(* CODESYS project SmiuUGP_Dubniki.project
   Version: 1.0
   Company: ENTEL

Project tree, tasks and I/O mapping:
  CODESYS_Control_for_Raspberry_Pi : CODESYS Control for Raspberry Pi, 3S - Smart Software Solutions GmbH, version 3.5.8.10
    application Application
      libraries: Util, * (System); AlarmManager, * (Intern); Alarm Manager Interfaces, * (Intern); Standard, * (System); VisuDialogs, * (System)
      task MainTask (cyclic, interval t#50ms, priority 2, watchdog t#1000ms x 1) calls PLC_PRG, GPIO_HANDLER, AlarmChecker
      task VISU_TASK (cyclic, interval 100 ms, priority 30) calls VisuElems.Visu_Prg
      task AlarmManagerTask (cyclic, interval 50 ms, priority 31) calls AlarmManager.Alarm_Prg
      task BusTask (cyclic, interval t#20ms, priority 1, watchdog t#1000ms x 1) calls BusReinit
      program PLC_PRG [ST]
      image pool ImagePool
      program GPIO_HANDLER [ST]
      visualization/
        visualisation monitoring
        ups_s2/
          visualisation ups_s2_state
          visualisation ups_s2_params
        visualisation main
        visualisation info
        visualisation climate
        visualisation alarm
        visualisation schrps
        visualisation shasn
        visualisation logs
        visualisation schrpa
        ups_s1/
          visualisation ups_s1_params
          visualisation ups_s1_state
        ups_a1/
          visualisation ups_a1_params
          visualisation ups_a1_state
        ups_a2/
          visualisation ups_a2_state
          visualisation ups_a2_params
        visualisation climate_log
        visualisation more
      Alarm Configuration
        alarm class Error (priority 10, acknowledge REP)
        alarm class Warning (priority 30, acknowledge REP)
        alarm class Info (priority 100, acknowledge REP)
        AlarmStorage
        text list AlarmGroup
        alarm group AlarmGroup
            93 [Error]: Comparison Equal, ExpressionToCompare TRUE, Expression AlarmChecker.ups_s2_out_v_alarm - "Отсутствует напряжение на выходе ИБП С2"
            94 [Error]: Comparison Equal, ExpressionToCompare TRUE, Expression AlarmChecker.ups_a1_out_v_alarm - "Отсутствует напряжение на выходе ИБП А1"
            49 [Error]: Comparison Equal, ExpressionToCompare TRUE, Expression PLC_PRG.ips_s1_alarm - "Авария ИБП С1"
            103 [Error]: Comparison Equal, ExpressionToCompare FALSE, Expression PLC_PRG.ips_s2_input_present - "ИБП С2 работает от АКБ"
            101 [Error]: Comparison Equal, ExpressionToCompare TRUE, Expression AlarmChecker.shrps_in_2_alarm - "Отсутствует напряжение на резервном вводе ЩРПС"
            97 [Error]: Comparison Equal, ExpressionToCompare TRUE, Expression GPIO_HANDLER.IN_1 - "Нарушение ШОС"
            100 [Error]: Comparison Equal, ExpressionToCompare TRUE, Expression AlarmChecker.shrps_in_1_alarm - "Отсутствует напряжение на основном вводе ЩРПC"
            92 [Error]: Comparison Equal, ExpressionToCompare TRUE, Expression AlarmChecker.ups_s1_out_v_alarm - "Отсутствует напряжение на выходе ИБП С1"
            95 [Error]: Comparison Equal, ExpressionToCompare TRUE, Expression AlarmChecker.ups_a2_out_v_alarm - "Отсутствует напряжение на выходе ИБП А2"
            47 [Error]: Comparison Equal, ExpressionToCompare TRUE, Expression PLC_PRG.ips_a2_alarm - "Авария ИБП А2"
            98 [Error]: Comparison Equal, ExpressionToCompare TRUE, Expression GPIO_HANDLER.IN_3 - "Авария ШОС"
            6 [Error]: Comparison Equal, ExpressionToCompare FALSE, Expression GPIO_HANDLER.IN_6 - "Отсутствует напряжение на шине БП ШАСН"
            90 [Error]: Comparison Equal, ExpressionToCompare TRUE, Expression AlarmChecker.ups_a1_in_v_alarm - "Отсутствует напряжение на входе ИБП А1"
            0 [Error]: Comparison Equal, ExpressionToCompare TRUE, Expression AlarmChecker.shrpa_in_1_alarm - "Отсутствует напряжение на основном вводе ЩРПА"
            1 [Error]: Comparison Equal, ExpressionToCompare TRUE, Expression AlarmChecker.shrpa_in_2_alarm - "Отсутствует напряжение на резервном вводе ЩРПА"
            2 [Error]: Comparison Equal, ExpressionToCompare FALSE, Expression GPIO_HANDLER.IN_4 - "Отсутствует напряжение на основном вводе ШАСН"
            3 [Error]: Comparison Equal, ExpressionToCompare FALSE, Expression GPIO_HANDLER.IN_5 - "Отсутствует напряжение на резервном вводе ШАСН"
            4 [Error]: Comparison Equal, ExpressionToCompare FALSE, Expression PLC_PRG.shrps_ups_bus_1 - "Отсутствует напряжение на ГП 1 ЩРПС"
            5 [Error]: Comparison Equal, ExpressionToCompare FALSE, Expression PLC_PRG.shrps_ups_bus_2 - "Отсутствует напряжение на ГП 2 ЩРПС"
            45 [Error]: Comparison Equal, ExpressionToCompare TRUE, Expression PLC_PRG.ips_a1_alarm - "Авария ИБП А1"
            102 [Error]: Comparison Equal, ExpressionToCompare FALSE, Expression PLC_PRG.ips_s1_input_present - "ИБП С1 работает от АКБ"
            88 [Error]: Comparison Equal, ExpressionToCompare TRUE, Expression AlarmChecker.ups_s1_in_v_alarm - "Отсутствует напряжение на входе ИБП С1"
            89 [Error]: Comparison Equal, ExpressionToCompare TRUE, Expression AlarmChecker.ups_s2_in_v_alarm - "Отсутствует напряжение на входе ИБП С2"
            99 [Error]: Comparison Equal, ExpressionToCompare TRUE, Expression AlarmChecker.shrpa_out_alarm - "Отсутствует напряжение на ШБПА  ЩРПА"
            91 [Error]: Comparison Equal, ExpressionToCompare TRUE, Expression AlarmChecker.ups_a2_in_v_alarm - "Отсутствует напряжение на входе ИБП А2"
            53 [Error]: Comparison Equal, ExpressionToCompare TRUE, Expression PLC_PRG.ips_s2_alarm - "Авария ИБП С2"
            96 [Error]: Comparison Equal, ExpressionToCompare TRUE, Expression GPIO_HANDLER.IN_2 - "Пожар"
            7 [Error]: Comparison Equal, ExpressionToCompare FALSE, Expression GPIO_HANDLER.IN_7 - "Отсутствует напряжение на шине ГП ШАСН"
        text list ClimateGroup
        alarm group ClimateGroup
            8 [Info]: Comparison Equal, ExpressionToCompare TRUE, Expression PLC_PRG.climate_condition_1_state - "Кондиционеры включены"
            11 [Info]: Comparison Equal, ExpressionToCompare FALSE, Expression PLC_PRG.climate_heat_door_state - "Обогрев дверей выключен"
            9 [Info]: Comparison Equal, ExpressionToCompare FALSE, Expression PLC_PRG.climate_condition_1_state - "Кондиционеры выключены"
            10 [Info]: Comparison Equal, ExpressionToCompare TRUE, Expression PLC_PRG.climate_heat_door_state - "Обогрев дверей включен"
            0 [Info]: Comparison Equal, ExpressionToCompare TRUE, Expression PLC_PRG.climate_heat_state - "Обогрев включен"
            1 [Info]: Comparison Equal, ExpressionToCompare TRUE, Expression PLC_PRG.climate_auto_state - "Автоматика включена"
            2 [Info]: Comparison Equal, ExpressionToCompare FALSE, Expression PLC_PRG.climate_heat_state - "Обогрев выключен"
            3 [Info]: Comparison Equal, ExpressionToCompare FALSE, Expression PLC_PRG.climate_auto_state - "Автоматика выключена"
            4 [Info]: Comparison Equal, ExpressionToCompare TRUE, Expression PLC_PRG.climate_zaslonka_state - "Заслонка открыта"
            5 [Info]: Comparison Equal, ExpressionToCompare FALSE, Expression PLC_PRG.climate_zaslonka_state - "Заслонка закрыта"
            6 [Info]: Comparison Equal, ExpressionToCompare TRUE, Expression PLC_PRG.climate_vent_1_state - "Вентиляторы включены"
            7 [Info]: Comparison Equal, ExpressionToCompare FALSE, Expression PLC_PRG.climate_vent_1_state - "Вентиляторы выключены"
            13 [Info]: Comparison Equal, ExpressionToCompare TRUE, Expression PLC_PRG.climate_temp_hight - "Высокая температура"
            12 [Info]: Comparison Equal, ExpressionToCompare TRUE, Expression PLC_PRG.climate_temp_low - "Низкая температура"
      program BusReinit [ST]
      program AlarmChecker [ST]
    SoftMotion General Axis Pool
    GPIOs_B_Pi2 : GPIOs B+/Pi2, 3S - Smart Software Solutions GmbH, version 1.1.1.10
        input  Application.GPIO_HANDLER.RAW_IN_10 : BOOL  // digital inputs (GPIO0..GPIO31).Bit5
        input  Application.GPIO_HANDLER.RAW_IN_12 : BOOL  // digital inputs (GPIO0..GPIO31).Bit6
        input  Application.GPIO_HANDLER.RAW_IN_9 : BOOL  // digital inputs (GPIO0..GPIO31).Bit7
        input  Application.GPIO_HANDLER.RAW_IN_8 : BOOL  // digital inputs (GPIO0..GPIO31).Bit8
        input  Application.GPIO_HANDLER.RAW_IN_3 : BOOL  // digital inputs (GPIO0..GPIO31).Bit10
        input  Application.GPIO_HANDLER.RAW_IN_11 : BOOL  // digital inputs (GPIO0..GPIO31).Bit12
        input  Application.GPIO_HANDLER.RAW_IN_1 : BOOL  // digital inputs (GPIO0..GPIO31).Bit13
        input  Application.GPIO_HANDLER.RAW_IN_6 : BOOL  // digital inputs (GPIO0..GPIO31).Bit18
        input  Application.GPIO_HANDLER.RAW_IN_7 : BOOL  // digital inputs (GPIO0..GPIO31).Bit21
        input  Application.GPIO_HANDLER.RAW_IN_5 : BOOL  // digital inputs (GPIO0..GPIO31).Bit23
        input  Application.GPIO_HANDLER.RAW_IN_4 : BOOL  // digital inputs (GPIO0..GPIO31).Bit24
        input  Application.GPIO_HANDLER.RAW_IN_2 : BOOL  // digital inputs (GPIO0..GPIO31).Bit25
        unmapped channels: digital inputs (GPIO0..GPIO31), digital outputs (GPIO0..GPIO31)
    Camera device
      <Empty>
    I²C
    SPI
    Onewire
    Ethernet : Ethernet, 3S - Smart Software Solutions GmbH, version 3.4.2.0
        settings: IPAddress = [192,168,10,200]; SubnetMask = [255,255,255,0]; GatewayAddress = [0,0,0,0]; NetworkInterfaceName = 'eth0'; NetworkInterfaceName = "eth0"
      Modbus_TCP_Master : Modbus TCP Master, 3S - Smart Software Solutions GmbH, version 3.5.4.0
          settings: AutoReconnect = TRUE
        IPS_2_2 : Modbus TCP Slave, 3S - Smart Software Solutions GmbH, version 3.5.4.0
            settings: Unit-ID = 1; ResponseTimeout = 1500; IPAddress = [192, 168, 10, 204]; Input_group.Function Code = 3; Input_group.Read Offset = 16#006D; Input_group.Read Length = 4; Input_group.Write Offset = 0; Input_group.Write Length = 0; Input_group.Cycle Time = 300; Output_group.Function Code = 3; Output_group.Read Offset = 16#0077; Output_group.Read Length = 7; Output_group.Write Offset = 0; Output_group.Write Length = 0; Output_group.Cycle Time = 300; Bypass_group.Function Code = 3; Bypass_group.Read Offset = 16#0081; Bypass_group.Read Length = 4; Bypass_group.Write Offset = 0; Bypass_group.Write Length = 0; Bypass_group.Cycle Time = 300; Battarey_group.Function Code = 3; Battarey_group.Read Offset = 16#0063; Battarey_group.Read Length = 4; Battarey_group.Write Offset = 0; Battarey_group.Write Length = 0; Battarey_group.Cycle Time = 300; Inv_Byp.Function Code = 3; Inv_Byp.Read Offset = 16#0095; Inv_Byp.Read Length = 1; Inv_Byp.Write Offset = 0; Inv_Byp.Write Length = 0; Inv_Byp.Cycle Time = 300; Status_group2.Function Code = 3; Status_group2.Read Offset = 16#0031; Status_group2.Read Length = 4; Status_group2.Write Offset = 0; Status_group2.Write Length = 0; Status_group2.Cycle Time = 300; Ivertor.Function Code = 3;
              Ivertor.Read Offset = 16#0096; Ivertor.Read Length = 1; Ivertor.Write Offset = 0; Ivertor.Write Length = 0; Ivertor.Cycle Time = 300; Battarey_temp.Function Code = 3; Battarey_temp.Read Offset = 16#001D; Battarey_temp.Read Length = 1; Battarey_temp.Write Offset = 0; Battarey_temp.Write Length = 0; Battarey_temp.Cycle Time = 300; Fault_grup.Function Code = 3; Fault_grup.Read Offset = 16#009F; Fault_grup.Read Length = 7; Fault_grup.Write Offset = 0; Fault_grup.Write Length = 0; Fault_grup.Cycle Time = 300
            input  Application.PLC_PRG.ips_s2_in_freq : WORD  // Input_group.Input_group
            input  Application.PLC_PRG.ips_s2_in_v_1 : WORD  // Input_group.Input_group
            input  Application.PLC_PRG.ips_s2_in_v_2 : WORD  // Input_group.Input_group
            input  Application.PLC_PRG.ips_s2_in_v_3 : WORD  // Input_group.Input_group
            input  Application.PLC_PRG.ips_s2_output_freq : WORD  // Output_group.Output_group
            input  Application.PLC_PRG.ips_s2_output_v_1 : WORD  // Output_group.Output_group
            input  Application.PLC_PRG.ips_s2_output_v_2 : WORD  // Output_group.Output_group
            input  Application.PLC_PRG.ips_s2_output_v_3 : WORD  // Output_group.Output_group
            input  Application.PLC_PRG.ips_s2_load_ph_1 : WORD  // Output_group.Output_group
            input  Application.PLC_PRG.ips_s2_load_ph_2 : WORD  // Output_group.Output_group
            input  Application.PLC_PRG.ips_s2_load_ph_3 : WORD  // Output_group.Output_group
            input  Application.PLC_PRG.ips_s2_bypass_freq : WORD  // Bypass_group.Bypass_group
            input  Application.PLC_PRG.ips_s2_bypass_v_1 : WORD  // Bypass_group.Bypass_group
            input  Application.PLC_PRG.ips_s2_bypass_v_2 : WORD  // Bypass_group.Bypass_group
            input  Application.PLC_PRG.ips_s2_bypass_v_3 : WORD  // Bypass_group.Bypass_group
            input  Application.PLC_PRG.ips_s2_battery_voltage : WORD  // Battarey_group.Battarey_group
            input  Application.PLC_PRG.ips_s2_battery_capacity : WORD  // Battarey_group.Battarey_group
            input  Application.PLC_PRG.ips_s2_time_m : WORD  // Battarey_group.Battarey_group
            input  Application.PLC_PRG.ips_s2_battery_current : WORD  // Battarey_group.Battarey_group
            input  Application.PLC_PRG.ips_s2_inv_byp : ARRAY[0..0] OF WORD  // Inv_Byp
            input  Application.PLC_PRG.ips_s2_state_reg : WORD  // Status_group2.Status_group2
            input  Application.PLC_PRG.ips_s2_Invertor : ARRAY[0..0] OF WORD  // Ivertor
            input  Application.PLC_PRG.ips_s2_temp : ARRAY[0..0] OF WORD  // Battarey_temp
            input  Application.PLC_PRG.ips_s2_emergency : WORD  // Fault_grup.Fault_grup
            input  Application.PLC_PRG.ips_s2_overload : WORD  // Fault_grup.Fault_grup
            input  Application.PLC_PRG.ips_s2_outfail : WORD  // Fault_grup.Fault_grup
            input  Application.PLC_PRG.ips_s2_overtemp : WORD  // Fault_grup.Fault_grup
            unmapped channels: Input_group, Output_group, Bypass_group, Battarey_group, Status_group2, Fault_grup
        IPS_2_1 : Modbus TCP Slave, 3S - Smart Software Solutions GmbH, version 3.5.4.0
            settings: Unit-ID = 1; ResponseTimeout = 1500; IPAddress = [192, 168, 10, 203]; Input_group.Function Code = 3; Input_group.Read Offset = 16#006D; Input_group.Read Length = 4; Input_group.Write Offset = 0; Input_group.Write Length = 0; Input_group.Cycle Time = 300; Output_group.Function Code = 3; Output_group.Read Offset = 16#0077; Output_group.Read Length = 7; Output_group.Write Offset = 0; Output_group.Write Length = 0; Output_group.Cycle Time = 300; Bypass_group.Function Code = 3; Bypass_group.Read Offset = 16#0081; Bypass_group.Read Length = 4; Bypass_group.Write Offset = 0; Bypass_group.Write Length = 0; Bypass_group.Cycle Time = 300; Battarey_group.Function Code = 3; Battarey_group.Read Offset = 16#0063; Battarey_group.Read Length = 4; Battarey_group.Write Offset = 0; Battarey_group.Write Length = 0; Battarey_group.Cycle Time = 300; Status2_group.Function Code = 3; Status2_group.Read Offset = 16#0031; Status2_group.Read Length = 4; Status2_group.Write Offset = 0; Status2_group.Write Length = 0; Status2_group.Cycle Time = 300; Invertor.Function Code = 3; Invertor.Read Offset = 16#0096; Invertor.Read Length = 1; Invertor.Write Offset = 0; Invertor.Write Length = 0; Invertor.Cycle Time = 300; Battarey_temp.Function Code = 3;
              Battarey_temp.Read Offset = 16#001D; Battarey_temp.Read Length = 1; Battarey_temp.Write Offset = 0; Battarey_temp.Write Length = 0; Battarey_temp.Cycle Time = 300; Inv_Byp.Function Code = 3; Inv_Byp.Read Offset = 16#0095; Inv_Byp.Read Length = 1; Inv_Byp.Write Offset = 0; Inv_Byp.Write Length = 0; Inv_Byp.Cycle Time = 300; Fault_group.Function Code = 3; Fault_group.Read Offset = 16#009F; Fault_group.Read Length = 7; Fault_group.Write Offset = 0; Fault_group.Write Length = 0; Fault_group.Cycle Time = 300
            input  Application.PLC_PRG.ips_s1_in_freq : WORD  // Input_group.Input_group
            input  Application.PLC_PRG.ips_s1_in_v_1 : WORD  // Input_group.Input_group
            input  Application.PLC_PRG.ips_s1_in_v_2 : WORD  // Input_group.Input_group
            input  Application.PLC_PRG.ips_s1_in_v_3 : WORD  // Input_group.Input_group
            input  Application.PLC_PRG.ips_s1_output_freq : WORD  // Output_group.Output_group
            input  Application.PLC_PRG.ips_s1_output_v_1 : WORD  // Output_group.Output_group
            input  Application.PLC_PRG.ips_s1_output_v_2 : WORD  // Output_group.Output_group
            input  Application.PLC_PRG.ips_s1_output_v_3 : WORD  // Output_group.Output_group
            input  Application.PLC_PRG.ips_s1_load_ph_1 : WORD  // Output_group.Output_group
            input  Application.PLC_PRG.ips_s1_load_ph_2 : WORD  // Output_group.Output_group
            input  Application.PLC_PRG.ips_s1_load_ph_3 : WORD  // Output_group.Output_group
            input  Application.PLC_PRG.ips_s1_bypass_freq : WORD  // Bypass_group.Bypass_group
            input  Application.PLC_PRG.ips_s1_bypass_v_1 : WORD  // Bypass_group.Bypass_group
            input  Application.PLC_PRG.ips_s1_bypass_v_2 : WORD  // Bypass_group.Bypass_group
            input  Application.PLC_PRG.ips_s1_bypass_v_3 : WORD  // Bypass_group.Bypass_group
            input  Application.PLC_PRG.ips_s1_battery_voltage : WORD  // Battarey_group.Battarey_group
            input  Application.PLC_PRG.ips_s1_battery_capacity : WORD  // Battarey_group.Battarey_group
            input  Application.PLC_PRG.ips_s1_time_m : WORD  // Battarey_group.Battarey_group
            input  Application.PLC_PRG.ips_s1_battery_current : WORD  // Battarey_group.Battarey_group
            input  Application.PLC_PRG.ips_s1_state_reg : WORD  // Status2_group.Status2_group
            input  Application.PLC_PRG.ips_s1_Invertor : ARRAY[0..0] OF WORD  // Invertor
            input  Application.PLC_PRG.ips_s1_temp : ARRAY[0..0] OF WORD  // Battarey_temp
            input  Application.PLC_PRG.ips_s1_inv_byp : ARRAY[0..0] OF WORD  // Inv_Byp
            input  Application.PLC_PRG.ips_s1_emergency : WORD  // Fault_group.Fault_group
            input  Application.PLC_PRG.ips_s1_overload : WORD  // Fault_group.Fault_group
            input  Application.PLC_PRG.ips_s1_outfail : WORD  // Fault_group.Fault_group
            input  Application.PLC_PRG.ips_s1_overtemp : WORD  // Fault_group.Fault_group
            unmapped channels: Input_group, Output_group, Bypass_group, Battarey_group, Status2_group, Fault_group
        IPS_1_1 : Modbus TCP Slave, 3S - Smart Software Solutions GmbH, version 3.5.4.0
            settings: Unit-ID = 1; ResponseTimeout = 1500; IPAddress = [192, 168, 10, 201]; Input_group.Function Code = 3; Input_group.Read Offset = 16#006D; Input_group.Read Length = 4; Input_group.Write Offset = 0; Input_group.Write Length = 0; Input_group.Cycle Time = 300; Output_group.Function Code = 3; Output_group.Read Offset = 16#0077; Output_group.Read Length = 5; Output_group.Write Offset = 0; Output_group.Write Length = 0; Output_group.Cycle Time = 300; Bypass_group.Function Code = 3; Bypass_group.Read Offset = 16#0081; Bypass_group.Read Length = 2; Bypass_group.Write Offset = 0; Bypass_group.Write Length = 0; Bypass_group.Cycle Time = 300; Battarey_group.Function Code = 3; Battarey_group.Read Offset = 16#0063; Battarey_group.Read Length = 4; Battarey_group.Write Offset = 0; Battarey_group.Write Length = 0; Battarey_group.Cycle Time = 300; Status_group2.Function Code = 3; Status_group2.Read Offset = 16#0031; Status_group2.Read Length = 4; Status_group2.Write Offset = 0; Status_group2.Write Length = 0; Status_group2.Cycle Time = 300; Invertor.Function Code = 3; Invertor.Read Offset = 16#0096; Invertor.Read Length = 1; Invertor.Write Offset = 0; Invertor.Write Length = 0; Invertor.Cycle Time = 300; Battarey_temp.Function Code = 3;
              Battarey_temp.Read Offset = 16#001D; Battarey_temp.Read Length = 1; Battarey_temp.Write Offset = 0; Battarey_temp.Write Length = 0; Battarey_temp.Cycle Time = 300; Inv_Byp.Function Code = 3; Inv_Byp.Read Offset = 16#0095; Inv_Byp.Read Length = 1; Inv_Byp.Write Offset = 0; Inv_Byp.Write Length = 0; Inv_Byp.Cycle Time = 300; Fault_group.Function Code = 3; Fault_group.Read Offset = 16#009F; Fault_group.Read Length = 7; Fault_group.Write Offset = 0; Fault_group.Write Length = 0; Fault_group.Cycle Time = 300
            input  Application.PLC_PRG.ips_a1_in_freq : WORD  // Input_group.Input_group
            input  Application.PLC_PRG.ips_a1_in_v_1 : WORD  // Input_group.Input_group
            input  Application.PLC_PRG.ips_a1_in_v_2 : WORD  // Input_group.Input_group
            input  Application.PLC_PRG.ips_a1_in_v_3 : WORD  // Input_group.Input_group
            input  Application.PLC_PRG.ips_a1_output_freq : WORD  // Output_group.Output_group
            input  Application.PLC_PRG.ips_a1_output_v_1 : WORD  // Output_group.Output_group
            input  Application.PLC_PRG.ips_a1_load_ph_1 : WORD  // Output_group.Output_group
            input  Application.PLC_PRG.ips_a1_bypass_freq : WORD  // Bypass_group.Bypass_group
            input  Application.PLC_PRG.ips_a1_bypass_v_1 : WORD  // Bypass_group.Bypass_group
            input  Application.PLC_PRG.ips_a1_battery_voltage : WORD  // Battarey_group.Battarey_group
            input  Application.PLC_PRG.ips_a1_battery_capacity : WORD  // Battarey_group.Battarey_group
            input  Application.PLC_PRG.ips_a1_time_m : WORD  // Battarey_group.Battarey_group
            input  Application.PLC_PRG.ips_a1_battery_current : WORD  // Battarey_group.Battarey_group
            input  Application.PLC_PRG.ips_a1_state_reg : WORD  // Status_group2.Status_group2
            input  Application.PLC_PRG.ips_a1_Invertor : ARRAY[0..0] OF WORD  // Invertor
            input  Application.PLC_PRG.ips_a1_temp : ARRAY[0..0] OF WORD  // Battarey_temp
            input  Application.PLC_PRG.ips_a1_inv_byp : ARRAY[0..0] OF WORD  // Inv_Byp
            input  Application.PLC_PRG.ips_a1_emergency : WORD  // Fault_group.Fault_group
            input  Application.PLC_PRG.ips_a1_overload : WORD  // Fault_group.Fault_group
            input  Application.PLC_PRG.ips_a1_outfail : WORD  // Fault_group.Fault_group
            input  Application.PLC_PRG.ips_a1_overtemp : WORD  // Fault_group.Fault_group
            unmapped channels: Input_group, Output_group, Bypass_group, Battarey_group, Status_group2, Fault_group
        IPS_1_2 : Modbus TCP Slave, 3S - Smart Software Solutions GmbH, version 3.5.4.0
            settings: Unit-ID = 1; ResponseTimeout = 1500; IPAddress = [192, 168, 10, 202]; Input_group.Function Code = 3; Input_group.Read Offset = 16#006D; Input_group.Read Length = 4; Input_group.Write Offset = 0; Input_group.Write Length = 0; Input_group.Cycle Time = 300; Output_group.Function Code = 3; Output_group.Read Offset = 16#0077; Output_group.Read Length = 5; Output_group.Write Offset = 0; Output_group.Write Length = 0; Output_group.Cycle Time = 300; Bypass_group.Function Code = 3; Bypass_group.Read Offset = 16#0081; Bypass_group.Read Length = 2; Bypass_group.Write Offset = 0; Bypass_group.Write Length = 0; Bypass_group.Cycle Time = 300; Battarey_group.Function Code = 3; Battarey_group.Read Offset = 16#0063; Battarey_group.Read Length = 4; Battarey_group.Write Offset = 0; Battarey_group.Write Length = 0; Battarey_group.Cycle Time = 300; Status_group2.Function Code = 3; Status_group2.Read Offset = 16#0031; Status_group2.Read Length = 4; Status_group2.Write Offset = 0; Status_group2.Write Length = 0; Status_group2.Cycle Time = 300; Invertor.Function Code = 3; Invertor.Read Offset = 16#0096; Invertor.Read Length = 1; Invertor.Write Offset = 0; Invertor.Write Length = 0; Invertor.Cycle Time = 300; Battarey_temp.Function Code = 3;
              Battarey_temp.Read Offset = 16#001D; Battarey_temp.Read Length = 1; Battarey_temp.Write Offset = 0; Battarey_temp.Write Length = 0; Battarey_temp.Cycle Time = 300; Inv_Byp.Function Code = 3; Inv_Byp.Read Offset = 16#0095; Inv_Byp.Read Length = 1; Inv_Byp.Write Offset = 0; Inv_Byp.Write Length = 0; Inv_Byp.Cycle Time = 300; Fault_group.Function Code = 3; Fault_group.Read Offset = 16#009F; Fault_group.Read Length = 7; Fault_group.Write Offset = 0; Fault_group.Write Length = 0; Fault_group.Cycle Time = 300
            input  Application.PLC_PRG.ips_a2_in_freq : WORD  // Input_group.Input_group
            input  Application.PLC_PRG.ips_a2_in_v_1 : WORD  // Input_group.Input_group
            input  Application.PLC_PRG.ips_a2_in_v_2 : WORD  // Input_group.Input_group
            input  Application.PLC_PRG.ips_a2_in_v_3 : WORD  // Input_group.Input_group
            input  Application.PLC_PRG.ips_a2_output_freq : WORD  // Output_group.Output_group
            input  Application.PLC_PRG.ips_a2_output_v_1 : WORD  // Output_group.Output_group
            input  Application.PLC_PRG.ips_a2_load_ph_1 : WORD  // Output_group.Output_group
            input  Application.PLC_PRG.ips_a2_bypass_freq : WORD  // Bypass_group.Bypass_group
            input  Application.PLC_PRG.ips_a2_bypass_v_1 : WORD  // Bypass_group.Bypass_group
            input  Application.PLC_PRG.ips_a2_battery_voltage : WORD  // Battarey_group.Battarey_group
            input  Application.PLC_PRG.ips_a2_battery_capacity : WORD  // Battarey_group.Battarey_group
            input  Application.PLC_PRG.ips_a2_time_m : WORD  // Battarey_group.Battarey_group
            input  Application.PLC_PRG.ips_a2_battery_current : WORD  // Battarey_group.Battarey_group
            input  Application.PLC_PRG.ips_a2_state_reg : WORD  // Status_group2.Status_group2
            input  Application.PLC_PRG.ips_a2_Invertor : ARRAY[0..0] OF WORD  // Invertor
            input  Application.PLC_PRG.ips_a2_temp : ARRAY[0..0] OF WORD  // Battarey_temp
            input  Application.PLC_PRG.ips_a2_inv_byp : ARRAY[0..0] OF WORD  // Inv_Byp
            input  Application.PLC_PRG.ips_a2_emergency : WORD  // Fault_group.Fault_group
            input  Application.PLC_PRG.ips_a2_overload : WORD  // Fault_group.Fault_group
            input  Application.PLC_PRG.ips_a2_outfail : WORD  // Fault_group.Fault_group
            input  Application.PLC_PRG.ips_a2_overtemp : WORD  // Fault_group.Fault_group
            unmapped channels: Input_group, Output_group, Bypass_group, Battarey_group, Status_group2, Fault_group
      ModbusTCP_Slave_Device : ModbusTCP Slave Device, 3S - Smart Software Solutions GmbH, version 3.5.5.0
          output Application.PLC_PRG.ips_s1_battery_capacity : WORD  // Outputs.Outputs
          output Application.PLC_PRG.ips_s1_battery_current : WORD  // Outputs.Outputs
          output Application.PLC_PRG.ips_s1_battery_time : WORD  // Outputs.Outputs
          output Application.PLC_PRG.ips_s1_battery_voltage : WORD  // Outputs.Outputs
          output Application.PLC_PRG.ips_s1_bypass_v_1 : WORD  // Outputs.Outputs
          output Application.PLC_PRG.ips_s1_bypass_v_2 : WORD  // Outputs.Outputs
          output Application.PLC_PRG.ips_s1_bypass_v_3 : WORD  // Outputs.Outputs
          output Application.PLC_PRG.ips_s1_in_v_1 : WORD  // Outputs.Outputs
          output Application.PLC_PRG.ips_s1_in_v_2 : WORD  // Outputs.Outputs
          output Application.PLC_PRG.ips_s1_in_v_3 : WORD  // Outputs.Outputs
          output Application.PLC_PRG.ips_s1_load_ph_1 : WORD  // Outputs.Outputs
          output Application.PLC_PRG.ips_s1_load_ph_2 : WORD  // Outputs.Outputs
          output Application.PLC_PRG.ips_s1_load_ph_3 : WORD  // Outputs.Outputs
          output Application.PLC_PRG.ips_s1_output_active_power_1 : WORD  // Outputs.Outputs
          output Application.PLC_PRG.ips_s1_output_active_power_2 : WORD  // Outputs.Outputs
          output Application.PLC_PRG.ips_s1_output_active_power_3 : WORD  // Outputs.Outputs
          output Application.PLC_PRG.ips_s1_output_freq : WORD  // Outputs.Outputs
          output Application.PLC_PRG.ips_s1_output_v_1 : WORD  // Outputs.Outputs
          output Application.PLC_PRG.ips_s1_output_v_2 : WORD  // Outputs.Outputs
          output Application.PLC_PRG.ips_s1_output_v_3 : WORD  // Outputs.Outputs
          output Application.PLC_PRG.ips_s1_temp : WORD  // Outputs.Outputs
          output Application.PLC_PRG.ips2_1_state : WORD  // Outputs.Outputs
          output Application.PLC_PRG.ips_s2_battery_capacity : WORD  // Outputs.Outputs
          output Application.PLC_PRG.ips_s2_battery_current : WORD  // Outputs.Outputs
          output Application.PLC_PRG.ips_s2_battery_time : WORD  // Outputs.Outputs
          output Application.PLC_PRG.ips_s2_battery_voltage : WORD  // Outputs.Outputs
          output Application.PLC_PRG.ips_s2_bypass_v_1 : WORD  // Outputs.Outputs
          output Application.PLC_PRG.ips_s2_bypass_v_2 : WORD  // Outputs.Outputs
          output Application.PLC_PRG.ips_s2_bypass_v_3 : WORD  // Outputs.Outputs
          output Application.PLC_PRG.ips_s2_in_v_1 : WORD  // Outputs.Outputs
          output Application.PLC_PRG.ips_s2_in_v_2 : WORD  // Outputs.Outputs
          output Application.PLC_PRG.ips_s2_in_v_3 : WORD  // Outputs.Outputs
          output Application.PLC_PRG.ips_s2_load_ph_1 : WORD  // Outputs.Outputs
          output Application.PLC_PRG.ips_s2_load_ph_2 : WORD  // Outputs.Outputs
          output Application.PLC_PRG.ips_s2_load_ph_3 : WORD  // Outputs.Outputs
          output Application.PLC_PRG.ips_s2_output_active_power_1 : WORD  // Outputs.Outputs
          output Application.PLC_PRG.ips_s2_output_active_power_2 : WORD  // Outputs.Outputs
          output Application.PLC_PRG.ips_s2_output_active_power_3 : WORD  // Outputs.Outputs
          output Application.PLC_PRG.ips_s2_output_freq : WORD  // Outputs.Outputs
          output Application.PLC_PRG.ips_s2_output_v_1 : WORD  // Outputs.Outputs
          output Application.PLC_PRG.ips_s2_output_v_2 : WORD  // Outputs.Outputs
          output Application.PLC_PRG.ips_s2_output_v_3 : WORD  // Outputs.Outputs
          output Application.PLC_PRG.ips_s2_temp : WORD  // Outputs.Outputs
          output Application.PLC_PRG.ips2_2_state : WORD  // Outputs.Outputs
          output Application.PLC_PRG.ips_a1_battery_capacity : WORD  // Outputs.Outputs
          output Application.PLC_PRG.ips_a1_battery_current : WORD  // Outputs.Outputs
          output Application.PLC_PRG.ips_a1_battery_time : WORD  // Outputs.Outputs
          output Application.PLC_PRG.ips_a1_battery_voltage : WORD  // Outputs.Outputs
          output Application.PLC_PRG.ips_a1_bypass_v_1 : WORD  // Outputs.Outputs
          output Application.PLC_PRG.ips_a1_in_v_1 : WORD  // Outputs.Outputs
          output Application.PLC_PRG.ips_a1_in_v_2 : WORD  // Outputs.Outputs
          output Application.PLC_PRG.ips_a1_in_v_3 : WORD  // Outputs.Outputs
          output Application.PLC_PRG.ips_a1_load_ph_1 : WORD  // Outputs.Outputs
          output Application.PLC_PRG.ips_a1_output_active_power_1 : WORD  // Outputs.Outputs
          output Application.PLC_PRG.ips_a1_output_freq : WORD  // Outputs.Outputs
          output Application.PLC_PRG.ips_a1_output_v_1 : WORD  // Outputs.Outputs
          output Application.PLC_PRG.ips_a1_temp : WORD  // Outputs.Outputs
          output Application.PLC_PRG.ips1_1_state : WORD  // Outputs.Outputs
          output Application.PLC_PRG.ips_a2_battery_capacity : WORD  // Outputs.Outputs
          output Application.PLC_PRG.ips_a2_battery_current : WORD  // Outputs.Outputs
          output Application.PLC_PRG.ips_a2_battery_time : WORD  // Outputs.Outputs
          output Application.PLC_PRG.ips_a2_battery_voltage : WORD  // Outputs.Outputs
          output Application.PLC_PRG.ips_a2_bypass_v_1 : WORD  // Outputs.Outputs
          output Application.PLC_PRG.ips_a2_in_v_1 : WORD  // Outputs.Outputs
          output Application.PLC_PRG.ips_a2_in_v_2 : WORD  // Outputs.Outputs
          output Application.PLC_PRG.ips_a2_in_v_3 : WORD  // Outputs.Outputs
          output Application.PLC_PRG.ips_a2_load_ph_1 : WORD  // Outputs.Outputs
          output Application.PLC_PRG.ips_a2_output_active_power_1 : WORD  // Outputs.Outputs
          output Application.PLC_PRG.ips_a2_output_freq : WORD  // Outputs.Outputs
          output Application.PLC_PRG.ips_a2_output_v_1 : WORD  // Outputs.Outputs
          output Application.PLC_PRG.ips_a2_temp : WORD  // Outputs.Outputs
          output Application.PLC_PRG.ips1_2_state : WORD  // Outputs.Outputs
          output Application.PLC_PRG.climate_state_reg : WORD  // Outputs.Outputs
          output Application.PLC_PRG.climate_temp_in : WORD  // Outputs.Outputs
          output Application.PLC_PRG.climate_temp_out : WORD  // Outputs.Outputs
          unmapped channels: Inputs, Outputs
    ModbusIN : Modbus COM, 3S - Smart Software Solutions GmbH, version 3.4.0.0
        settings: DataBits = 8; StopBits = 1; ComPort = 1
      ModbusMaster : Modbus Master, COM Port, 3S - Smart Software Solutions GmbH, version 3.5.5.0
          settings: Transmission = 'RTU'; ResponseTimeout = 60; TimeBetweenFrames = 20; Auto-restart communication = TRUE
        PLC : Modbus Slave, COM Port, 3S - Smart Software Solutions GmbH, version 3.5.4.0
            settings: SlaveAddress = 1; ResponseTimeout = 100; UseExtendedFunctionCodes = TRUE; Channel 0.Function Code = 3; Channel 0.Read Offset = 16#EB28; Channel 0.Read Length = 3; Channel 0.Write Offset = 0; Channel 0.Write Length = 0; Channel 0.Cycle Time = 500
            input  Application.PLC_PRG.climate_temp_in : WORD  // Channel 0.Channel 0
            input  Application.PLC_PRG.climate_temp_out : WORD  // Channel 0.Channel 0
            input  Application.PLC_PRG.climate_state_reg : WORD  // Channel 0.Channel 0
            unmapped channels: Channel 0
        SHRPA_ICP_CON : Modbus Slave, COM Port, 3S - Smart Software Solutions GmbH, version 3.5.4.0
            settings: SlaveAddress = 101; ResponseTimeout = 50; UseExtendedFunctionCodes = TRUE; DI.Function Code = 2; DI.Read Offset = 16#0000; DI.Read Length = 16; DI.Write Offset = 0; DI.Write Length = 0; DI.Cycle Time = 100
            input  Application.PLC_PRG.shrpa_in_1 : BOOL  // DI.DI.Bit0
            input  Application.PLC_PRG.shrpa_in_2 : BOOL  // DI.DI.Bit1
            input  Application.PLC_PRG.shrpa_ups_in_1_raw : BOOL  // DI.DI.Bit2
            input  Application.PLC_PRG.shrpa_ups_in_2_raw : BOOL  // DI.DI.Bit3
            input  Application.PLC_PRG.shrpa_input_switch_state_1 : BOOL  // DI.DI.Bit4
            input  Application.PLC_PRG.shrpa_input_switch_state_2 : BOOL  // DI.DI.Bit5
            input  Application.PLC_PRG.shrpa_ups_out_1 : BOOL  // DI.DI.Bit6
            input  Application.PLC_PRG.shrpa_ups_out_2 : BOOL  // DI.DI.Bit7
            input  Application.PLC_PRG.shrpa_load_line_1_source_state_1 : BOOL  // DI.DI.Bit0
            input  Application.PLC_PRG.shrpa_load_line_1_source_state_2 : BOOL  // DI.DI.Bit1
            input  Application.PLC_PRG.shrpa_load_line_2_source_state_2 : BOOL  // DI.DI.Bit2
            input  Application.PLC_PRG.shrpa_load_line_2_source_state_1 : BOOL  // DI.DI.Bit3
            input  Application.PLC_PRG.shrpa_input_tv1 : BOOL  // DI.DI.Bit4
            input  Application.PLC_PRG.shrpa_bypass_in_1 : BOOL  // DI.DI.Bit5
            input  Application.PLC_PRG.shrpa_bypass_in_2 : BOOL  // DI.DI.Bit6
            unmapped channels: DI
        SHRPS_ICP_CON : Modbus Slave, COM Port, 3S - Smart Software Solutions GmbH, version 3.5.4.0
            settings: SlaveAddress = 102; ResponseTimeout = 50; UseExtendedFunctionCodes = TRUE; DI.Function Code = 2; DI.Read Offset = 16#0000; DI.Read Length = 16; DI.Write Offset = 0; DI.Write Length = 0; DI.Cycle Time = 100
            input  Application.PLC_PRG.shrps_in_1 : BOOL  // DI.DI.Bit0
            input  Application.PLC_PRG.shrps_in_2 : BOOL  // DI.DI.Bit1
            input  Application.PLC_PRG.shrps_ups_in_1 : BOOL  // DI.DI.Bit2
            input  Application.PLC_PRG.shrps_bypass_in_1 : BOOL  // DI.DI.Bit3
            input  Application.PLC_PRG.shrps_ups_in_2 : BOOL  // DI.DI.Bit4
            input  Application.PLC_PRG.shrps_bypass_in_2 : BOOL  // DI.DI.Bit5
            input  Application.PLC_PRG.shrps_ups_out_1 : BOOL  // DI.DI.Bit6
            input  Application.PLC_PRG.shrps_ups_out_2 : BOOL  // DI.DI.Bit7
            input  Application.PLC_PRG.shrps_bypass_out : BOOL  // DI.DI.Bit0
            input  Application.PLC_PRG.shrps_ups_bus_1_raw : BOOL  // DI.DI.Bit1
            input  Application.PLC_PRG.shrps_ups_bus_2_raw : BOOL  // DI.DI.Bit2
            unmapped channels: DI
        SHASN_ICP_CON : Modbus Slave, COM Port, 3S - Smart Software Solutions GmbH, version 3.5.4.0
            settings: SlaveAddress = 103; ResponseTimeout = 50; UseExtendedFunctionCodes = TRUE; DI.Function Code = 2; DI.Read Offset = 16#0000; DI.Read Length = 16; DI.Write Offset = 0; DI.Write Length = 0; DI.Cycle Time = 100
            unmapped channels: DI
        SHRPA_ELNET_2 : Modbus Slave, COM Port, 3S - Smart Software Solutions GmbH, version 3.5.4.0
            settings: SlaveAddress = 12; ResponseTimeout = 100; UseExtendedFunctionCodes = TRUE; Voltage.Function Code = 3; Voltage.Read Offset = 16#0001; Voltage.Read Length = 6; Voltage.Write Offset = 0; Voltage.Write Length = 0; Voltage.Cycle Time = 500; Current.Function Code = 3; Current.Read Offset = 16#000D; Current.Read Length = 6; Current.Write Offset = 0; Current.Write Length = 0; Current.Cycle Time = 500
            input  Application.PLC_PRG.shrpa_voltage_registers2 : ARRAY[0..5] OF WORD  // Voltage
            unmapped channels: Current
        SHRPA_ELNET_1 : Modbus Slave, COM Port, 3S - Smart Software Solutions GmbH, version 3.5.4.0
            settings: SlaveAddress = 11; ResponseTimeout = 100; UseExtendedFunctionCodes = TRUE; Voltage.Function Code = 3; Voltage.Read Offset = 16#0001; Voltage.Read Length = 6; Voltage.Write Offset = 0; Voltage.Write Length = 0; Voltage.Cycle Time = 500; Current.Function Code = 3; Current.Read Offset = 16#000D; Current.Read Length = 6; Current.Write Offset = 0; Current.Write Length = 0; Current.Cycle Time = 500
            input  Application.PLC_PRG.shrpa_voltage_registers1 : ARRAY[0..5] OF WORD  // Voltage
            unmapped channels: Current
        SHRPA_ELNET_3 : Modbus Slave, COM Port, 3S - Smart Software Solutions GmbH, version 3.5.4.0
            settings: SlaveAddress = 13; ResponseTimeout = 100; UseExtendedFunctionCodes = TRUE; Voltage.Function Code = 3; Voltage.Read Offset = 16#0001; Voltage.Read Length = 2; Voltage.Write Offset = 0; Voltage.Write Length = 0; Voltage.Cycle Time = 500; Current.Function Code = 3; Current.Read Offset = 16#000D; Current.Read Length = 2; Current.Write Offset = 0; Current.Write Length = 0; Current.Cycle Time = 500; Freq.Function Code = 3; Freq.Read Offset = 16#0033; Freq.Read Length = 2; Freq.Write Offset = 0; Freq.Write Length = 0; Freq.Cycle Time = 500
            input  Application.PLC_PRG.shrpa_voltage_registers3 : ARRAY[0..1] OF WORD  // Voltage
            input  Application.PLC_PRG.shrpa_current_registers3 : ARRAY[0..1] OF WORD  // Current
            input  Application.PLC_PRG.shrpa_freq_registers3 : ARRAY[0..1] OF WORD  // Freq
        SHRPA_ELNET_4 : Modbus Slave, COM Port, 3S - Smart Software Solutions GmbH, version 3.5.4.0
            settings: SlaveAddress = 14; ResponseTimeout = 100; UseExtendedFunctionCodes = TRUE; Voltage.Function Code = 3; Voltage.Read Offset = 16#0001; Voltage.Read Length = 2; Voltage.Write Offset = 0; Voltage.Write Length = 0; Voltage.Cycle Time = 500; Current.Function Code = 3; Current.Read Offset = 16#000D; Current.Read Length = 2; Current.Write Offset = 0; Current.Write Length = 0; Current.Cycle Time = 500; Freq.Function Code = 3; Freq.Read Offset = 16#0033; Freq.Read Length = 2; Freq.Write Offset = 0; Freq.Write Length = 0; Freq.Cycle Time = 500
            input  Application.PLC_PRG.shrpa_voltage_registers4 : ARRAY[0..1] OF WORD  // Voltage
            input  Application.PLC_PRG.shrpa_current_registers4 : ARRAY[0..1] OF WORD  // Current
            input  Application.PLC_PRG.shrpa_freq_registers4 : ARRAY[0..1] OF WORD  // Freq
        SHRPS_ELNET_1 : Modbus Slave, COM Port, 3S - Smart Software Solutions GmbH, version 3.5.4.0
            settings: SlaveAddress = 21; ResponseTimeout = 100; UseExtendedFunctionCodes = TRUE; Voltage.Function Code = 3; Voltage.Read Offset = 16#0001; Voltage.Read Length = 6; Voltage.Write Offset = 0; Voltage.Write Length = 0; Voltage.Cycle Time = 500; Current.Function Code = 3; Current.Read Offset = 16#000D; Current.Read Length = 6; Current.Write Offset = 0; Current.Write Length = 0; Current.Cycle Time = 500
            input  Application.PLC_PRG.shrps_voltage_registers1 : ARRAY[0..5] OF WORD  // Voltage
            unmapped channels: Current
        SHRPS_ELNET_2 : Modbus Slave, COM Port, 3S - Smart Software Solutions GmbH, version 3.5.4.0
            settings: SlaveAddress = 22; ResponseTimeout = 100; UseExtendedFunctionCodes = TRUE; Voltage.Function Code = 3; Voltage.Read Offset = 16#0001; Voltage.Read Length = 6; Voltage.Write Offset = 0; Voltage.Write Length = 0; Voltage.Cycle Time = 500; Current.Function Code = 3; Current.Read Offset = 16#000D; Current.Read Length = 6; Current.Write Offset = 0; Current.Write Length = 0; Current.Cycle Time = 500
            input  Application.PLC_PRG.shrps_voltage_registers2 : ARRAY[0..5] OF WORD  // Voltage
            unmapped channels: Current
        SHRPS_ELNET_3 : Modbus Slave, COM Port, 3S - Smart Software Solutions GmbH, version 3.5.4.0
            settings: SlaveAddress = 23; ResponseTimeout = 100; UseExtendedFunctionCodes = TRUE; Voltage.Function Code = 3; Voltage.Read Offset = 16#0001; Voltage.Read Length = 6; Voltage.Write Offset = 0; Voltage.Write Length = 0; Voltage.Cycle Time = 500; Current.Function Code = 3; Current.Read Offset = 16#000D; Current.Read Length = 6; Current.Write Offset = 0; Current.Write Length = 0; Current.Cycle Time = 500
            input  Application.PLC_PRG.shrps_voltage_registers3 : ARRAY[0..5] OF WORD  // Voltage
            unmapped channels: Current
        SHRPS_ELNET_4 : Modbus Slave, COM Port, 3S - Smart Software Solutions GmbH, version 3.5.4.0
            settings: SlaveAddress = 24; ResponseTimeout = 100; UseExtendedFunctionCodes = TRUE; Voltage.Function Code = 3; Voltage.Read Offset = 16#0001; Voltage.Read Length = 6; Voltage.Write Offset = 0; Voltage.Write Length = 0; Voltage.Cycle Time = 500; Current.Function Code = 3; Current.Read Offset = 16#000D; Current.Read Length = 6; Current.Write Offset = 0; Current.Write Length = 0; Current.Cycle Time = 500
            input  Application.PLC_PRG.shrps_voltage_registers4 : ARRAY[0..5] OF WORD  // Voltage
            unmapped channels: Current
  text list GlobalTextList
  5ce3da45-db07-42e7-a21c-a00fff4ed8f6|Images\bg_800.png
  5ce3da45-db07-42e7-a21c-a00fff4ed8f6|Images\mpx_state_bg.png
  5ce3da45-db07-42e7-a21c-a00fff4ed8f6|Images\ups\bypass_line_on.png
  5ce3da45-db07-42e7-a21c-a00fff4ed8f6|Images\ups\bypass_line_off.png
  5ce3da45-db07-42e7-a21c-a00fff4ed8f6|Images\ups\battery_arrow_off.png
  5ce3da45-db07-42e7-a21c-a00fff4ed8f6|Images\ups\battery_arrow_on.png
  5ce3da45-db07-42e7-a21c-a00fff4ed8f6|Images\ups\battery_line_off.png
  5ce3da45-db07-42e7-a21c-a00fff4ed8f6|Images\ups\battery_line_on.png
  5ce3da45-db07-42e7-a21c-a00fff4ed8f6|Images\ups\bypass_arrow_off.png
  5ce3da45-db07-42e7-a21c-a00fff4ed8f6|Images\ups\bypass_arrow_on.png
  5ce3da45-db07-42e7-a21c-a00fff4ed8f6|Images\ups\arrow_off.png
  5ce3da45-db07-42e7-a21c-a00fff4ed8f6|Images\ups\arrow_on.png
  5ce3da45-db07-42e7-a21c-a00fff4ed8f6|C:\workspace\SmiuUGP\Images\Proba.png
  5ce3da45-db07-42e7-a21c-a00fff4ed8f6|C:\workspace\SmiuUGP\Images\main_bg.png
  5ce3da45-db07-42e7-a21c-a00fff4ed8f6|C:\workspace\SmiuUGP\Images\bg_800.png
  5ce3da45-db07-42e7-a21c-a00fff4ed8f6|E:\YandexDisk\Скриншоты\ups.png
  5ce3da45-db07-42e7-a21c-a00fff4ed8f6|C:\workspace\SmiuUGP\Images\mpx_state_bg.png
  5ce3da45-db07-42e7-a21c-a00fff4ed8f6|C:\workspace\SmiuUGP\Images\scheme.png
  5ce3da45-db07-42e7-a21c-a00fff4ed8f6|C:\workspace\SmiuUGP\Images\more_info.png
  5ce3da45-db07-42e7-a21c-a00fff4ed8f6|C:\workspace\SmiuUGP\Images\log.png
  5ce3da45-db07-42e7-a21c-a00fff4ed8f6|C:\workspace\SmiuUGP\Images\gpio_1.png
  5ce3da45-db07-42e7-a21c-a00fff4ed8f6|release_images\schrpa.png
  5ce3da45-db07-42e7-a21c-a00fff4ed8f6|C:\workspace\SmiuUGP\Images\volt.png
  5ce3da45-db07-42e7-a21c-a00fff4ed8f6|release_images\shasn.png
  5ce3da45-db07-42e7-a21c-a00fff4ed8f6|C:\workspace\SmiuUGP\Images\battery.png
  5ce3da45-db07-42e7-a21c-a00fff4ed8f6|C:\workspace\SmiuUGP\Images\climate.png
  5ce3da45-db07-42e7-a21c-a00fff4ed8f6|C:\workspace\SmiuUGP\Images\alert.png
  5ce3da45-db07-42e7-a21c-a00fff4ed8f6|C:\workspace\SmiuUGP\Images\automation.png
  5ce3da45-db07-42e7-a21c-a00fff4ed8f6|E:\SmiuLinux\smiu_logo.png
  5ce3da45-db07-42e7-a21c-a00fff4ed8f6|C:\workspace\SmiuUGP\Images\mini_ups.png
  5ce3da45-db07-42e7-a21c-a00fff4ed8f6|release_images\shrpa.png
  5ce3da45-db07-42e7-a21c-a00fff4ed8f6|release_images\schrps.png
  5ce3da45-db07-42e7-a21c-a00fff4ed8f6|C:\workspace\UGP\Dubniki_03_2016\Images\shrpa.png
*)

// CODESYS_Control_for_Raspberry_Pi/Application/PLC_PRG
PROGRAM PLC_PRG
VAR	
	//----------------- Визуализация -----------------//
	var_true :BOOL := TRUE;
	ack		 :BOOL;
	history  :BOOL;	
	

	//----------------- ЩРПА -----------------//
	// ICP CON
	shrpa_in_1                       : BOOL; // ЩРПА ввод 1 - состояние автомата
	shrpa_in_2                       : BOOL; // ЩРПА ввод 2 - состояние автомата
	shrpa_ups_in_1_raw               : BOOL; // ввод ИБП А1 (инвертировано)
	shrpa_ups_in_2_raw               : BOOL; // ввод ИБП А2 (инвертировано)	
	shrpa_ups_in_1                   : BOOL; // ввод ИБП А1
	shrpa_ups_in_2                   : BOOL; // ввод ИБП А2
	shrpa_input_switch_state_1       : BOOL; // QS1 в  1 положениии
	shrpa_input_switch_state_2       : BOOL; // QS1 во 2 положениии
	shrpa_ups_out_1                  : BOOL; // ЩРПА ИБП А1 - выход (состояние автомата)
	shrpa_ups_out_2                  : BOOL; // ЩРПА ИБП А2 - выход (состояние автомата)
	shrpa_load_line_1_source_state_1 : BOOL; // QS2  в 1 положении
	shrpa_load_line_1_source_state_2 : BOOL; // QS2 во 2 положении
	shrpa_load_line_2_source_state_1 : BOOL; // QS3  в 1 положении
	shrpa_load_line_2_source_state_2 : BOOL; // QS3 во 2 положении
	shrpa_input_tv1                  : BOOL; // ЩРПА Трансформатор - выход (состояние автомата)
	shrpa_bypass_in_1                : BOOL; // ЩРПА ИБП А1 - байпас (состояние автомата)
	shrpa_bypass_in_2                : BOOL; // ЩРПА ИБП А2 - байпас (состояние автомата)
	
	//ELNET
	delay_timeout 			    : TIME := T#6S; // Таймаут ошибки связи
	
	shrpa_voltage_registers1    : ARRAY [1..6] OF WORD; 
	shrpa_voltage_registers2    : ARRAY [1..6] OF WORD;
	shrpa_voltage_registers3    : ARRAY [1..2] OF WORD;
	shrpa_voltage_registers4    : ARRAY [1..2] OF WORD;
	
	shrpa_current_registers3    : ARRAY [1..2] OF WORD;
	shrpa_current_registers4    : ARRAY [1..2] OF WORD;
	
	shrpa_freq_registers3       : ARRAY [1..2] OF WORD;
	shrpa_freq_registers4       : ARRAY [1..2] OF WORD;
	
	shrpa_voltage_1_delay_timer	: TON;
	shrpa_voltage_2_delay_timer	: TON;
	shrpa_voltage_3_delay_timer	: TON;
	shrpa_voltage_4_delay_timer	: TON;
	
	shrpa_voltage_1_sum_checker : REAL;
	shrpa_voltage_2_sum_checker : REAL;
	
	shrpa_voltage_1_line_1      : REAL; // ЩРПА ELNET#1 - V L1 
	shrpa_voltage_1_line_2      : REAL;	// ЩРПА ELNET#1 - V L2
	shrpa_voltage_1_line_3      : REAL;	// ЩРПА ELNET#1 - V L3
	
	shrpa_voltage_2_line_1      : REAL;	// ЩРПА ELNET#2 - V L1
	shrpa_voltage_2_line_2      : REAL;	// ЩРПА ELNET#2 - V L2
	shrpa_voltage_2_line_3      : REAL;	// ЩРПА ELNET#2 - V L3
	
	shrpa_voltage_3_line_1      : REAL;	// ЩРПА ELNET#3 - V L1
	shrpa_voltage_4_line_1      : REAL; // ЩРПА ELNET#4 - V L1
	
	shrpa_current_3_line_1      : REAL;	// ЩРПА ELNET#3 - I L1
	shrpa_current_4_line_1      : REAL; // ЩРПА ELNET#4 - I L1
	
	shrpa_freq_3_line_1         : REAL;	// ЩРПА ELNET#3 - F L1
	shrpa_freq_4_line_1         : REAL; // ЩРПА ELNET#4 - F L1

	
	//----------------- ЩРПС -----------------//
	// ICP CON
	shrps_in_1          : BOOL; // ЩРПС ввод 1 - состояние автомата
	shrps_in_2          : BOOL;	// ЩРПС ввод 2 - состояние автомата
	shrps_ups_in_1      : BOOL;	// ИБП C1 - ввод (состояние автомата)
	shrps_ups_in_2      : BOOL;	// ИБП C2 - ввод (состояние автомата)		
	shrps_bypass_in_1   : BOOL;	// ИБП С1 - байпас
	shrps_bypass_in_2   : BOOL;	// ИБП C2 - байпас
	shrps_ups_out_1     : BOOL;	// ИБП C1 - выход
	shrps_ups_out_2     : BOOL;	// ИБП C2 - выход
	shrps_bypass_out    : BOOL;	// ЩРПС - байпас шины 
	shrps_ups_bus_1_raw : BOOL; // ЩРПС БП#1 - наличие напряжения (инвертировано)
	shrps_ups_bus_2_raw : BOOL;	// ЩРПС БП#2 - наличие напряжения (инвертировано)
	shrps_ups_bus_1     : BOOL; // ЩРПС БП#1 - наличие напряжения
	shrps_ups_bus_2     : BOOL; // ЩРПС БП#2 - наличие напряжения
		
	//ELNET
	shrps_voltage_registers1 : ARRAY [1..6] OF WORD;
	shrps_voltage_registers2 : ARRAY [1..6] OF WORD;
	shrps_voltage_registers3 : ARRAY [1..6] OF WORD;
	shrps_voltage_registers4 : ARRAY [1..6] OF WORD;
	
	shrps_voltage_1_delay_timer	: TON;
	shrps_voltage_2_delay_timer	: TON;
	shrps_voltage_3_delay_timer	: TON;
	shrps_voltage_4_delay_timer	: TON;
	
	shrps_voltage_1_sum_checker : REAL;
	shrps_voltage_2_sum_checker : REAL;
	shrps_voltage_3_sum_checker : REAL;
	shrps_voltage_4_sum_checker : REAL;

	shrps_voltage_1_line_1 : REAL; // ЩРПС ELNET#1 - V L1 
	shrps_voltage_1_line_2 : REAL; // ЩРПС ELNET#1 - V L2
	shrps_voltage_1_line_3 : REAL; // ЩРПС ELNET#1 - V L3
	
	shrps_voltage_2_line_1 : REAL; // ЩРПС ELNET#2 - V L1 
	shrps_voltage_2_line_2 : REAL; // ЩРПС ELNET#2 - V L2 
	shrps_voltage_2_line_3 : REAL; // ЩРПС ELNET#2 - V L3
	
	shrps_voltage_3_line_1 : REAL; // ЩРПС ELNET#3 - V L1 
	shrps_voltage_3_line_2 : REAL; // ЩРПС ELNET#3 - V L2 
	shrps_voltage_3_line_3 : REAL; // ЩРПС ELNET#3 - V L3
	
	shrps_voltage_4_line_1 : REAL; // ЩРПС ELNET#4 - V L1 
	shrps_voltage_4_line_2 : REAL; // ЩРПС ELNET#4 - V L2 
	shrps_voltage_4_line_3 : REAL; // ЩРПА ELNET#4 - V L3 


	//----------------- Климат -----------------//	
	climate_temp_out          :WORD; 
	climat_temp_out_minus     :BOOL; // Бит отрицательности температуры
	climate_temp_out_real     :REAL; // Наружная температура
	climate_temp_in           :WORD; 
	climat_temp_in_minus      :BOOL; // Бит отрицательности температуры
	climate_temp_in_real      :REAL; // Внутренняя температура
	climate_state_reg         :WORD; 
	climate_state_as_bit      :WORD_AS_BIT;
	climate_zaslonka_state    :BOOL; // Состояние заслонки
	climate_vent_1_state      :BOOL; // Состояние вентилятора №1
	climate_vent_2_state      :BOOL; // Состояние вентилятора №2
	climate_condition_1_state :BOOL; // Состояние кондиционера №1
	climate_condition_2_state :BOOL; // Состояние кондиционера №2
	climate_heat_state        :BOOL; // Состояние обогрева
	climate_heat_door_state   :BOOL; // Состояние обогрева дверей
	climate_auto_state        :BOOL; // Состояние автоматики климата
	climate_temp_excess       :BOOL; // авария. внутренняя температура > 25
	climate_temp_hight		  :BOOL; // 12 бит Высокая температура
	climate_temp_low		  :BOOL; // 11 бит Низкая температура
	
	
	//----------------- ИБП А1 (IPS) -----------------//	
	ips_a1_power					  :WORD := 40; // Мощность ИБП в кВт
	ips_a1_cosphi                     :REAL := 0.83; // Cos phi
	ips_a1_time_m					  :WORD; // Время автономии в мин
	ips_a1_in_v_1 	 		   		  :WORD; // 1-е Напряжение входа
	ips_a1_in_v_2 	 		   		  :WORD; // 2-e Напряжение входа
	ips_a1_in_v_3 	 		   		  :WORD; // 3-е Напряжение входа
	ips_a1_in_v_1_real 	 		   	  :REAL; // 1-е Напряжение входа (x0.1)
	ips_a1_in_v_2_real 	 		   	  :REAL; // 2-e Напряжение входа (x0.1)
	ips_a1_in_v_3_real 	 		   	  :REAL; // 3-е Напряжение входа (x0.1)
	ips_a1_in_freq 	 		   		  :WORD; // Частота на входе
	ips_a1_in_freq_real		   		  :REAL; // Частота на входе (x0.1)
	ips_a1_bypass_v_1  		   		  :WORD; // 1-е Напряжение байпаса
	ips_a1_bypass_v_1_real  		  :REAL; // 1-е Напряжение байпаса (x0.1)
	ips_a1_bypass_freq 		   		  :WORD; // Частота байпаса
	ips_a1_bypass_freq_real      	  :REAL; // Частота байпаса
	ips_a1_output_v_1  		   		  :WORD; // 1-е Напряжение выхода
	ips_a1_output_v_1_real  		  :REAL; // 1-е Напряжение выхода (x0.1)
	ips_a1_output_active_power_1      :WORD; // Активная мощность 1-й фазы (кВт)
	ips_a1_output_active_power_1_real :REAL; // Активная мощность 1-й фазы (кВт)
	ips_a1_output_freq 	       		  :WORD; // Частота выхода
	ips_a1_output_freq_real 	      :REAL; // Частота выхода (x0.1)
	ips_a1_load_ph_1    	       	  :WORD; // Загрузска 1-й фазы (%)
	ips_a1_load_ph_1_real    	      :REAL; // Загрузска 1-й фазы (%) (x0.1)
	ips_a1_battery_voltage 	   		  :WORD; // Напряжение батареи
	ips_a1_battery_voltage_real  	  :REAL; // Напряжение батареи (x0.1)
	ips_a1_battery_current 	   		  :WORD; // Ток батареи
	ips_a1_battery_current_real  	  :REAL; // Ток батареи (x0.1)
	ips_a1_battery_capacity 	   	  :WORD; // Остаточная емкость батареи (%)
	ips_a1_battery_time 		   	  :WORD; // Остаточное время автономии (минуты)
	ips_a1_temp 				   	  :WORD; // Температура
	ips_a1_temp_real				  :REAL; // Температура (x0.1)
	
	ips_a1_invertor  				  :WORD; // Работа от инвертора (14 = ДА, 16 = НЕТ)	
	ips_a1_state_reg 	       		  :WORD; // Регистр состояния#1 (2 = От сети (Байпас), 3 = АКБП (Байпас))
	ips_a1_inv_byp					  :WORD; // Регистр состояния#2 (13 = Байпас) 

	//Переменные для отображения состояния ИБП
	ips_a1_bypass_line_state 	   	  :STRING; 
	ips_a1_bypass_arrow_state         :STRING;
	ips_a1_battery_arrow_state 		  :STRING; // Состояние батареи
	ips_a1_battery_line_state 		  :STRING; // Состояние батареи
	ips_a1_input_state 		   		  :STRING; // Состояние входа
	ips_a1_output_state 		   	  :STRING; // Состояние выхода
	ips_a1_arrow_state 				  :STRING;
	ips_a1_alarm                      :BOOL;   // Общая авария
	ips_a1_overtemp					  :WORD;   // Превышена температура (14 = ДА)
	ips_a1_overload					  :WORD;   // Перегрузка (14 = ДА)
	ips_a1_outfail					  :WORD;   //
	ips_a1_emergency				  :WORD;   // 

	
	//----------------- ИБП А2 (IPS) -----------------//	
	ips_a2_power					  :WORD := 40; // Мощность ИБП в кВт
	ips_a2_cosphi                     :REAL := 0.83; // Cos phi
	ips_a2_time_m					  :WORD; // Время автономии в мин
	ips_a2_in_v_1 	 		   		  :WORD; // 1-е Напряжение входа
	ips_a2_in_v_2 	 		   		  :WORD; // 2-e Напряжение входа
	ips_a2_in_v_3 	 		   		  :WORD; // 3-е Напряжение входа
	ips_a2_in_v_1_real 	 		   	  :REAL; // 1-е Напряжение входа (x0.1)
	ips_a2_in_v_2_real 	 		   	  :REAL; // 2-e Напряжение входа (x0.1)
	ips_a2_in_v_3_real 	 		   	  :REAL; // 3-е Напряжение входа (x0.1)
	ips_a2_in_freq 	 		   		  :WORD; // Частота на входе
	ips_a2_in_freq_real		   		  :REAL; // Частота на входе (x0.1)
	ips_a2_bypass_v_1  		   		  :WORD; // 1-е Напряжение байпаса
	ips_a2_bypass_v_1_real  		  :REAL; // 1-е Напряжение байпаса (x0.1)
	ips_a2_bypass_freq 		   		  :WORD; // Частота байпаса
	ips_a2_bypass_freq_real      	  :REAL; // Частота байпаса
	ips_a2_output_v_1  		   		  :WORD; // 1-е Напряжение выхода
	ips_a2_output_v_1_real  		  :REAL; // 1-е Напряжение выхода (x0.1)
	ips_a2_output_active_power_1      :WORD; // Активная мощность 1-й фазы (кВт)
	ips_a2_output_active_power_1_real :REAL; // Активная мощность 1-й фазы (кВт)
	ips_a2_output_freq 	       		  :WORD; // Частота выхода
	ips_a2_output_freq_real 	      :REAL; // Частота выхода (x0.1)
	ips_a2_load_ph_1    	       	  :WORD; // Загрузска 1-й фазы (%)
	ips_a2_load_ph_1_real    	      :REAL; // Загрузска 1-й фазы (%) (x0.1)
	ips_a2_battery_voltage 	   		  :WORD; // Напряжение батареи
	ips_a2_battery_voltage_real  	  :REAL; // Напряжение батареи (x0.1)
	ips_a2_battery_current 	   		  :WORD; // Ток батареи
	ips_a2_battery_current_real  	  :REAL; // Ток батареи (x0.1)
	ips_a2_battery_capacity 	   	  :WORD; // Остаточная емкость батареи (%)
	ips_a2_battery_time 		   	  :WORD; // Остаточное время автономии (минуты)
	ips_a2_temp 				   	  :WORD; // Температура
	ips_a2_temp_real				  :REAL; // Температура (x0.1)
	
	ips_a2_invertor  				  :WORD; // Работа от инвертора (14 = ДА, 16 = НЕТ)	
	ips_a2_state_reg 	       		  :WORD; // Регистр состояния#1 (2 = От сети (Байпас), 3 = АКБП (Байпас))
	ips_a2_inv_byp					  :WORD; // Регистр состояния#2 (13 = Байпас) 

	//Переменные для отображения состояния ИБП
	ips_a2_bypass_line_state 	   	  :STRING; 
	ips_a2_bypass_arrow_state         :STRING;
	ips_a2_battery_arrow_state 		  :STRING; // Состояние батареи
	ips_a2_battery_line_state 		  :STRING; // Состояние батареи
	ips_a2_input_state 		   		  :STRING; // Состояние входа
	ips_a2_output_state 		   	  :STRING; // Состояние выхода
	ips_a2_arrow_state 				  :STRING;
	ips_a2_alarm                      :BOOL;   // Общая авария
	ips_a2_overtemp					  :WORD;   // Превышена температура (14 = ДА)
	ips_a2_overload					  :WORD;   // Перегрузка (14 = ДА)
	ips_a2_outfail					  :WORD;   //
	ips_a2_emergency				  :WORD;   // 
	
	//----------------- ИБП С1 (IPS) -----------------//	
	ips_s1_power				      :WORD := 150;	//Мощность ИБП в кВт
	ips_s1_cosphi                     :REAL := 0.83; // Cos phi
	ips_s1_time_m					  :WORD; // Время автономии в мин
	ips_s1_in_v_1 	 		   		  :WORD; // 1-е Напрядение входа
	ips_s1_in_v_2 	 		   		  :WORD; // 2-e Напряжение входа
	ips_s1_in_v_3 	 		   		  :WORD; // 3-е Напряжение входа
	ips_s1_in_v_1_real 	 		   	  :REAL; // 1-е Напрядение входа (x0.1)
	ips_s1_in_v_2_real 	 		   	  :REAL; // 2-e Напряжение входа (x0.1)
	ips_s1_in_v_3_real 	 		   	  :REAL; // 3-е Напряжение входа (x0.1)
	ips_s1_in_freq 	 		   		  :WORD; // Частота на входе
	ips_s1_in_freq_real		   		  :REAL; // Частота на входе (x0.1)
	ips_s1_bypass_v_1  		   		  :WORD; // 1-е Напряжение байпаса
	ips_s1_bypass_v_2  		   		  :WORD; // 2-е Напряжение байпаса
	ips_s1_bypass_v_3  		   		  :WORD; // 3-е Напряжение байпаса
	ips_s1_bypass_v_1_real  		  :REAL; // 1-е Напряжение байпаса (x0.1)
	ips_s1_bypass_v_2_real  		  :REAL; // 2-е Напряжение байпаса (x0.1)
	ips_s1_bypass_v_3_real  		  :REAL; // 3-е Напряжение байпаса (x0.1)
	ips_s1_bypass_freq 		   		  :WORD; // Частота байпаса
	ips_s1_bypass_freq_real      	  :REAL; // Частота байпаса
	ips_s1_output_v_1  		   		  :WORD; // 1-е Напряжение выхода
	ips_s1_output_v_2  		   		  :WORD; // 2-е Напряжение выхода
	ips_s1_output_v_3  		   		  :WORD; // 3-е Напряжение выхода
	ips_s1_output_v_1_real  		  :REAL; // 1-е Напряжение выхода (x0.1)
	ips_s1_output_v_2_real  		  :REAL; // 2-е Напряжение выхода (x0.1)
	ips_s1_output_v_3_real  		  :REAL; // 3-е Напряжение выхода (x0.1)
	ips_s1_output_active_power_1	  :WORD; // Активная мощность - L1
	ips_s1_output_active_power_2	  :WORD; // Активная мощность - L2
	ips_s1_output_active_power_3	  :WORD; // Активная мощность - L2
	ips_s1_output_active_power_1_real :REAL; //Активная мощность 1-й фазы (кВт)
	ips_s1_output_active_power_2_real :REAL; //Активная мощность 2-й фазы (кВт)
	ips_s1_output_active_power_3_real :REAL; //Активная мощность 3-й фазы (кВт)
	ips_s1_output_active_power_real   :REAL; //Активная мощность всех фаз
	ips_s1_output_freq 	       		  :WORD; //Частота выхода
	ips_s1_output_freq_real 	      :REAL; //Частота выхода (x0.1)
	ips_s1_load_ph_1    	       	  :WORD; //Загрузска 1-й фазы (%)
	ips_s1_load_ph_2    		   	  :WORD; //Загрузска 3-й фазы (%)
	ips_s1_load_ph_3    	       	  :WORD; //Загрузска 2-й фазы (%)
	ips_s1_load_ph_1_real    	      :REAL; //Загрузска 1-й фазы (%) (x0.1)
	ips_s1_load_ph_2_real    		  :REAL; //Загрузска 3-й фазы (%) (x0.1)
	ips_s1_load_ph_3_real    	      :REAL; //Загрузска 2-й фазы (%) (x0.1)
	ips_s1_battery_voltage 	   		  :WORD; //Напряжение батареи
	ips_s1_battery_voltage_real  	  :REAL; //Напряжение батареи (x0.1)
	ips_s1_battery_current 	   		  :WORD; //Ток батареи
	ips_s1_battery_current_real  	  :REAL; //Ток батареи (x0.1)
	ips_s1_battery_capacity 	      :WORD; //Остаточная емкость батареи (%)
	ips_s1_battery_time 		   	  :WORD; //Остаточное время автономии (минуты)
	ips_s1_temp 				   	  :WORD; //Температура
	ips_s1_temp_real				  :REAL; //Температура (x0.1)
	
	ips_s1_invertor  				  :WORD; // Работа от инвертора (14 = ДА, 16 = НЕТ)	
	ips_s1_state_reg 	       		  :WORD; // Регистр состояния#1 (2 = От сети (Байпас), 3 = АКБП (Байпас))
	ips_s1_inv_byp					  :WORD; // Регистр состояния#2 (13 = Байпас) 

	//Переменные для отображения состояния ИБП
	ips_s1_bypass_line_state 	   	  :STRING; 
	ips_s1_bypass_arrow_state    	  :STRING;
	ips_s1_battery_arrow_state 		  :STRING; // Состояние батареи
	ips_s1_battery_line_state 		  :STRING; // Состояние батареи
	ips_s1_input_state 		   		  :STRING; // Состояние входа
	ips_s1_output_state 		   	  :STRING; // Состояние выхода
	ips_s1_arrow_state 				  :STRING;
	ips_s1_alarm                      :BOOL;   // Общая авария
	ips_s1_overtemp					  :WORD;   // Превышена температура (14 = ДА)
	ips_s1_overload					  :WORD;   // Перегрузка (14 = ДА)
	ips_s1_outfail					  :WORD;   //
	ips_s1_emergency				  :WORD;   //
	
	ips_s1_input_present              :BOOL;   // Наличиче напряжения на входе
	

	//----------------- ИБП С2 (IPS) -----------------//	
	ips_s2_power				      :WORD := 150;	//Мощность ИБП в кВт
	ips_s2_cosphi                     :REAL := 0.83; // Cos phi
	ips_s2_time_m					  :WORD; // Время автономии в мин
	ips_s2_in_v_1 	 		   		  :WORD; // 1-е Напрядение входа
	ips_s2_in_v_2 	 		   		  :WORD; // 2-e Напряжение входа
	ips_s2_in_v_3 	 		   		  :WORD; // 3-е Напряжение входа
	ips_s2_in_v_1_real 	 		   	  :REAL; // 1-е Напрядение входа (x0.1)
	ips_s2_in_v_2_real 	 		   	  :REAL; // 2-e Напряжение входа (x0.1)
	ips_s2_in_v_3_real 	 		   	  :REAL; // 3-е Напряжение входа (x0.1)
	ips_s2_in_freq 	 		   		  :WORD; // Частота на входе
	ips_s2_in_freq_real		   		  :REAL; // Частота на входе (x0.1)
	ips_s2_bypass_v_1  		   		  :WORD; // 1-е Напряжение байпаса
	ips_s2_bypass_v_2  		   		  :WORD; // 2-е Напряжение байпаса
	ips_s2_bypass_v_3  		   		  :WORD; // 3-е Напряжение байпаса
	ips_s2_bypass_v_1_real  		  :REAL; // 1-е Напряжение байпаса (x0.1)
	ips_s2_bypass_v_2_real  		  :REAL; // 2-е Напряжение байпаса (x0.1)
	ips_s2_bypass_v_3_real  		  :REAL; // 3-е Напряжение байпаса (x0.1)
	ips_s2_bypass_freq 		   		  :WORD; // Частота байпаса
	ips_s2_bypass_freq_real      	  :REAL; // Частота байпаса
	ips_s2_output_v_1  		   		  :WORD; // 1-е Напряжение выхода
	ips_s2_output_v_2  		   		  :WORD; // 2-е Напряжение выхода
	ips_s2_output_v_3  		   		  :WORD; // 3-е Напряжение выхода
	ips_s2_output_v_1_real  		  :REAL; // 1-е Напряжение выхода (x0.1)
	ips_s2_output_v_2_real  		  :REAL; // 2-е Напряжение выхода (x0.1)
	ips_s2_output_v_3_real  		  :REAL; // 3-е Напряжение выхода (x0.1)
	ips_s2_output_active_power_1	  :WORD; // Активная мощность - L1
	ips_s2_output_active_power_2	  :WORD; // Активная мощность - L2
	ips_s2_output_active_power_3	  :WORD; // Активная мощность - L2
	ips_s2_output_active_power_1_real :REAL; //Активная мощность 1-й фазы (кВт)
	ips_s2_output_active_power_2_real :REAL; //Активная мощность 2-й фазы (кВт)
	ips_s2_output_active_power_3_real :REAL; //Активная мощность 3-й фазы (кВт)
	ips_s2_output_active_power_real   :REAL; //Активная мощность всех фаз
	ips_s2_output_freq 	       		  :WORD; //Частота выхода
	ips_s2_output_freq_real 	      :REAL; //Частота выхода (x0.1)
	ips_s2_load_ph_1    	       	  :WORD; //Загрузска 1-й фазы (%)
	ips_s2_load_ph_2    		   	  :WORD; //Загрузска 3-й фазы (%)
	ips_s2_load_ph_3    	       	  :WORD; //Загрузска 2-й фазы (%)
	ips_s2_load_ph_1_real    	      :REAL; //Загрузска 1-й фазы (%) (x0.1)
	ips_s2_load_ph_2_real    		  :REAL; //Загрузска 3-й фазы (%) (x0.1)
	ips_s2_load_ph_3_real    	      :REAL; //Загрузска 2-й фазы (%) (x0.1)
	ips_s2_battery_voltage 	   		  :WORD; //Напряжение батареи
	ips_s2_battery_voltage_real  	  :REAL; //Напряжение батареи (x0.1)
	ips_s2_battery_current 	   		  :WORD; //Ток батареи
	ips_s2_battery_current_real  	  :REAL; //Ток батареи (x0.1)
	ips_s2_battery_capacity 	      :WORD; //Остаточная емкость батареи (%)
	ips_s2_battery_time 		   	  :WORD; //Остаточное время автономии (минуты)
	ips_s2_temp 				   	  :WORD; //Температура
	ips_s2_temp_real				  :REAL; //Температура (x0.1)
	
	ips_s2_invertor  				  :WORD; // Работа от инвертора (14 = ДА, 16 = НЕТ)	
	ips_s2_state_reg 	       		  :WORD; // Регистр состояния#1 (2 = От сети (Байпас), 3 = АКБП (Байпас))
	ips_s2_inv_byp					  :WORD; // Регистр состояния#2 (13 = Байпас) 

	//Переменные для отображения состояния ИБП
	ips_s2_bypass_line_state 	   	  :STRING; 
	ips_s2_bypass_arrow_state    	  :STRING;
	ips_s2_battery_arrow_state 		  :STRING; // Состояние батареи
	ips_s2_battery_line_state 		  :STRING; // Состояние батареи
	ips_s2_input_state 		   		  :STRING; // Состояние входа
	ips_s2_output_state 		   	  :STRING; // Состояние выхода
	ips_s2_arrow_state 				  :STRING;
	ips_s2_alarm                      :BOOL;   // Общая авария
	ips_s2_overtemp					  :WORD;   // Превышена температура (14 = ДА)
	ips_s2_overload					  :WORD;   // Перегрузка (14 = ДА)
	ips_s2_outfail					  :WORD;   //
	ips_s2_emergency				  :WORD;   //
	
	ips_s2_input_present              :BOOL;   // Наличиче напряжения на входе
	
	//---------------------------------------------------------------
	ips1_1_state						:WORD;
	ips1_2_state						:WORD;
	ips2_1_state						:WORD;
	ips2_2_state						:WORD;
	
	mpx_s1_state_string :WSTRING := "";
	mpx_s2_state_string :WSTRING := "";
	mpx_a1_state_string :WSTRING := "";
	mpx_a2_state_string :WSTRING := "";
	
END_VAR

// Работа с ICP CON
shrps_ups_bus_1 := NOT(shrps_ups_bus_1_raw);
shrps_ups_bus_2 := NOT(shrps_ups_bus_2_raw);
shrpa_ups_in_1 := NOT(shrpa_ups_in_1_raw);
shrpa_ups_in_2 := NOT(shrpa_ups_in_2_raw);

// Работа с ElNet
// ЩРПА
shrpa_voltage_1_sum_checker := shrpa_voltage_registers1[2] + shrpa_voltage_registers1[4] + shrpa_voltage_registers1[6];
Shrpa_voltage_1_delay_timer(IN := (shrpa_voltage_1_sum_checker = 0), PT:= delay_timeout);
IF (Shrpa_voltage_1_delay_timer.Q = TRUE) THEN
	shrpa_voltage_1_line_1 := 0;
	shrpa_voltage_1_line_2 := 0;
	shrpa_voltage_1_line_3 := 0;
ELSIF (shrpa_voltage_1_sum_checker > 0) THEN
	shrpa_voltage_1_line_1 := shrpa_voltage_registers1[2];
	shrpa_voltage_1_line_2 := shrpa_voltage_registers1[4];
	shrpa_voltage_1_line_3 := shrpa_voltage_registers1[6];
END_IF

shrpa_voltage_2_sum_checker := shrpa_voltage_registers2[2] + shrpa_voltage_registers2[4] + shrpa_voltage_registers2[6];
Shrpa_voltage_2_delay_timer(IN := (shrpa_voltage_2_sum_checker = 0), PT:= delay_timeout);
IF (Shrpa_voltage_2_delay_timer.Q = TRUE) THEN
	shrpa_voltage_2_line_1 := 0;
	shrpa_voltage_2_line_2 := 0;
	shrpa_voltage_2_line_3 := 0;
ELSIF (shrpa_voltage_2_sum_checker > 0) THEN
	shrpa_voltage_2_line_1 := shrpa_voltage_registers2[2];
	shrpa_voltage_2_line_2 := shrpa_voltage_registers2[4];
	shrpa_voltage_2_line_3 := shrpa_voltage_registers2[6];
END_IF

Shrpa_voltage_3_delay_timer(IN := (shrpa_voltage_registers3[2] = 0), PT:= delay_timeout);
IF (Shrpa_voltage_3_delay_timer.Q = TRUE) THEN
	shrpa_voltage_3_line_1 := 0;
	shrpa_current_3_line_1 := 0;
	shrpa_freq_3_line_1 := 0;
ELSIF (shrpa_voltage_registers3[2] > 0) THEN
	shrpa_voltage_3_line_1 := shrpa_voltage_registers3[2];
	shrpa_current_3_line_1 := shrpa_current_registers3[2];
	shrpa_freq_3_line_1 := shrpa_freq_registers3[2];
END_IF

Shrpa_voltage_4_delay_timer(IN := (shrpa_voltage_registers4[2] = 0), PT:= delay_timeout);
IF (Shrpa_voltage_4_delay_timer.Q = TRUE) THEN
	shrpa_voltage_4_line_1 := 0;
	shrpa_current_4_line_1 := 0;
	shrpa_freq_4_line_1 := 0;
ELSIF (shrpa_voltage_registers4[2] > 0) THEN
	shrpa_voltage_4_line_1 := shrpa_voltage_registers4[2];
	shrpa_current_4_line_1 := shrpa_current_registers4[2];
	shrpa_freq_4_line_1 := shrpa_freq_registers4[2];
END_IF

// ЩРПС
shrps_voltage_1_sum_checker := shrps_voltage_registers1[2] + shrps_voltage_registers1[4] + shrps_voltage_registers1[6];
Shrps_voltage_1_delay_timer(IN := (shrps_voltage_1_sum_checker = 0), PT:= delay_timeout);
IF (Shrps_voltage_1_delay_timer.Q = TRUE) THEN
	shrps_voltage_1_line_1 := 0;
	shrps_voltage_1_line_2 := 0;
	shrps_voltage_1_line_3 := 0;
ELSIF (shrps_voltage_1_sum_checker > 0) THEN
	shrps_voltage_1_line_1 := shrps_voltage_registers1[2];
	shrps_voltage_1_line_2 := shrps_voltage_registers1[4];
	shrps_voltage_1_line_3 := shrps_voltage_registers1[6];
END_IF

shrps_voltage_2_sum_checker := shrps_voltage_registers2[2] + shrps_voltage_registers2[4] + shrps_voltage_registers2[6];
Shrps_voltage_2_delay_timer(IN := (shrps_voltage_2_sum_checker = 0), PT:= delay_timeout);
IF (Shrps_voltage_2_delay_timer.Q = TRUE) THEN
	shrps_voltage_2_line_1 := 0;
	shrps_voltage_2_line_2 := 0;
	shrps_voltage_2_line_3 := 0;
ELSIF (shrps_voltage_2_sum_checker > 0) THEN
	shrps_voltage_2_line_1 := shrps_voltage_registers2[2];
	shrps_voltage_2_line_2 := shrps_voltage_registers2[4];
	shrps_voltage_2_line_3 := shrps_voltage_registers2[6];
END_IF

shrps_voltage_3_sum_checker := shrps_voltage_registers3[2] + shrps_voltage_registers3[4] + shrps_voltage_registers3[6];
Shrps_voltage_3_delay_timer(IN := (shrps_voltage_3_sum_checker = 0), PT:= delay_timeout);
IF (Shrps_voltage_3_delay_timer.Q = TRUE) THEN
	shrps_voltage_3_line_1 := 0;
	shrps_voltage_3_line_2 := 0;
	shrps_voltage_3_line_3 := 0;
ELSIF (shrps_voltage_3_sum_checker > 0) THEN
	shrps_voltage_3_line_1 := shrps_voltage_registers3[2];
	shrps_voltage_3_line_2 := shrps_voltage_registers3[4];
	shrps_voltage_3_line_3 := shrps_voltage_registers3[6];
END_IF

shrps_voltage_4_sum_checker := shrps_voltage_registers4[2] + shrps_voltage_registers4[4] + shrps_voltage_registers4[6];
Shrps_voltage_4_delay_timer(IN := (shrps_voltage_4_sum_checker = 0), PT:= delay_timeout);
IF (Shrps_voltage_4_delay_timer.Q = TRUE) THEN
	shrps_voltage_4_line_1 := 0;
	shrps_voltage_4_line_2 := 0;
	shrps_voltage_4_line_3 := 0;
ELSIF (shrps_voltage_4_sum_checker > 0) THEN
	shrps_voltage_4_line_1 := shrps_voltage_registers4[2];
	shrps_voltage_4_line_2 := shrps_voltage_registers4[4];
	shrps_voltage_4_line_3 := shrps_voltage_registers4[6];
END_IF

//Работа с климатом
climate_state_as_bit(W    := climate_state_reg);
climate_zaslonka_state    := climate_state_as_bit.B03;
climate_vent_1_state      := climate_state_as_bit.B00;
climate_vent_2_state      := climate_state_as_bit.B01;
climate_condition_1_state := climate_state_as_bit.B04;
climate_condition_2_state := climate_state_as_bit.B05;
climate_heat_state        := climate_state_as_bit.B02;
climate_heat_door_state   := climate_state_as_bit.B06;
climate_auto_state        := NOT(climate_state_as_bit.B07);
climat_temp_out_minus     := climate_state_as_bit.B10;
climat_temp_in_minus      := climate_state_as_bit.B09;
climate_temp_low      	  := climate_state_as_bit.B11;
climate_temp_hight        := climate_state_as_bit.B12;

climate_temp_out_real     := climate_temp_out * 0.1;
climate_temp_in_real      := climate_temp_in * 0.1;
IF (climat_temp_out_minus = TRUE) THEN
	climate_temp_out_real := climate_temp_out_real * (-1);
END_IF
IF (climat_temp_in_minus = TRUE) THEN
	climate_temp_in_real := climate_temp_in_real * (-1);
END_IF
IF (climate_temp_in_real > 25) THEN
	climate_temp_excess := TRUE;
	ELSE
		climate_temp_excess := FALSE;
END_IF

//------------------------------------ИБП A1 (IPS)-------------------------------------
//Конвертация параметров IPS 1.1
ips_a1_in_v_1_real 	 		   	:= ips_a1_in_v_1 * 0.1;
ips_a1_in_v_2_real 	 			:= ips_a1_in_v_2 * 0.1;   		
ips_a1_in_v_3_real 	 		 	:= ips_a1_in_v_3 * 0.1;  		
ips_a1_in_freq_real               := ips_a1_in_freq * 0.1;

ips_a1_bypass_v_1_real			:= ips_a1_bypass_v_1 * 0.1;
ips_a1_bypass_freq_real           := ips_a1_bypass_freq * 0.1;

ips_a1_output_v_1_real			:= ips_a1_output_v_1 * 0.1;
ips_a1_output_freq_real           := ips_a1_output_freq * 0.1;

ips_a1_load_ph_1_real				:= ips_a1_load_ph_1 * 0.1;
ips_a1_output_active_power_1_real	:= ips_a1_power * ips_a1_load_ph_1_real * 0.01 * ips_a1_cosphi;

ips_a1_output_active_power_1 		:= REAL_TO_WORD(ips_a1_output_active_power_1_real * 1000);

ips_a1_battery_voltage_real       := ips_a1_battery_voltage * 1;
ips_a1_battery_current_real       := ips_a1_battery_current * 0.1;

ips_a1_temp_real 					:= ips_a1_temp * 0.1;


//Логика состояний IPS 1.1
IF ((ips_a1_Invertor = 14) AND (ips_a1_state_reg = 2) AND (ips_a1_inv_byp = 12)) THEN
	ips_a1_bypass_line_state := 'bypass_line1_off';
	ips_a1_bypass_arrow_state := 'bypass_arrow_off';
	ips_a1_input_state := 'arrow_on';	
	ips_a1_output_state := 'arrow_on';
	ips_a1_arrow_state := 'arrow_on';
	ips_a1_battery_line_state := 'battery_line_on';
	ips_a1_battery_arrow_state := 'battery_arrow_on';
	mpx_a1_state_string := "От сети";	
	ips1_1_state := 1;
ELSE
	IF ((ips_a1_Invertor = 14) AND (ips_a1_state_reg = 3) AND (ips_a1_inv_byp = 12)) THEN	
		ips_a1_bypass_line_state := 'bypass_line1_off';
		ips_a1_bypass_arrow_state := 'bypass_arrow_off';
		ips_a1_input_state := 'arrow_off';
		ips_a1_output_state := 'arrow_on';
		ips_a1_arrow_state := 'arrow_on';
		ips_a1_battery_line_state := 'battery_line_on';
		ips_a1_battery_arrow_state := 'battery_arrow_on';
		mpx_a1_state_string := "От АКБ";
		ips1_1_state := 2;	
	ELSE	
		IF ((ips_a1_Invertor = 16) AND (ips_a1_state_reg = 3) AND (ips_a1_inv_byp = 13)) THEN	
			ips_a1_bypass_line_state := 'bypass_line_on';
			ips_a1_bypass_arrow_state := 'bypass_arrow_on';
			ips_a1_input_state := 'arrow_off';
			ips_a1_output_state := 'arrow_on';
			ips_a1_arrow_state := 'arrow_off';
			ips_a1_battery_line_state := 'battery_line_off';
			ips_a1_battery_arrow_state := 'battery_arrow_off';
			mpx_a1_state_string := "Байпас";
			ips1_1_state := 3;	
		ELSE	
			IF ((ips_a1_Invertor = 14) AND (ips_a1_state_reg = 2) AND (ips_a1_inv_byp = 13)) THEN	
				ips_a1_bypass_line_state := 'bypass_line_on';
				ips_a1_bypass_arrow_state := 'bypass_arrow_on';
				ips_a1_input_state := 'arrow_off';
				ips_a1_output_state := 'arrow_on';
				ips_a1_arrow_state := 'arrow_off';
				ips_a1_battery_line_state := 'battery_line_off';
				ips_a1_battery_arrow_state := 'battery_arrow_off';
				mpx_a1_state_string := "Байпас";
				ips1_1_state := 3;	
			ELSE	
				ips_a1_bypass_line_state := 'bypass_line1_off';
				ips_a1_bypass_arrow_state := 'bypass_arrow_off';
				ips_a1_input_state := 'arrow_off';
				ips_a1_output_state := 'arrow_off';
				ips_a1_arrow_state := 'arrow_off';
				ips_a1_battery_line_state := 'battery_line_off';
				ips_a1_battery_arrow_state := 'battery_arrow_off';
				mpx_a1_state_string := "Неизвестно";
				ips1_1_state := 0;
			END_IF
		END_IF
	END_IF
END_IF

IF ((ips_a1_overtemp = 14) OR (ips_a1_overload = 14) OR (ips_a1_outfail = 14) OR (ips_a1_emergency = 14)) THEN
	ips_a1_alarm := TRUE;
ELSE
	ips_a1_alarm := FALSE;
END_IF

//------------------------------------IPS 1.2-------------------------------------
//Конвертация параметров IPS 1.2
ips_a2_in_v_1_real 	 		   	:= ips_a2_in_v_1 * 0.1;
ips_a2_in_v_2_real 	 			:= ips_a2_in_v_2 * 0.1;   		
ips_a2_in_v_3_real 	 		 	:= ips_a2_in_v_3 * 0.1;  		
ips_a2_in_freq_real               := ips_a2_in_freq * 0.1;

ips_a2_bypass_v_1_real			:= ips_a2_bypass_v_1 * 0.1;
ips_a2_bypass_freq_real           := ips_a2_bypass_freq * 0.1;

ips_a2_output_v_1_real			:= ips_a2_output_v_1 * 0.1;
ips_a2_output_freq_real           := ips_a2_output_freq * 0.1;

ips_a2_load_ph_1_real				:= ips_a2_load_ph_1 * 0.1;
ips_a2_output_active_power_1_real	:= ips_a2_power * ips_a2_load_ph_1_real * 0.01 * ips_a2_cosphi;

ips_a2_output_active_power_1 		:= REAL_TO_WORD(ips_a2_output_active_power_1_real * 1000);

ips_a2_battery_voltage_real       := ips_a2_battery_voltage * 1;
ips_a2_battery_current_real       := ips_a2_battery_current * 0.1;

ips_a2_temp_real 					:= ips_a2_temp * 0.1;


//Логика состояний IPS 1.2
IF ((ips_a2_Invertor = 14) AND (ips_a2_state_reg = 2) AND (ips_a2_inv_byp = 12)) THEN
	ips_a2_bypass_line_state := 'bypass_line1_off';
	ips_a2_bypass_arrow_state := 'bypass_arrow_off';
	ips_a2_input_state := 'arrow_on';	
	ips_a2_output_state := 'arrow_on';
	ips_a2_arrow_state := 'arrow_on';
	ips_a2_battery_line_state := 'battery_line_on';
	ips_a2_battery_arrow_state := 'battery_arrow_on';
	mpx_a2_state_string := "От сети";	
	ips1_2_state := 1;
ELSE
	IF ((ips_a2_Invertor = 14) AND (ips_a2_state_reg = 3) AND (ips_a2_inv_byp = 12)) THEN	
		ips_a2_bypass_line_state := 'bypass_line1_off';
		ips_a2_bypass_arrow_state := 'bypass_arrow_off';
		ips_a2_input_state := 'arrow_off';
		ips_a2_output_state := 'arrow_on';
		ips_a2_arrow_state := 'arrow_on';
		ips_a2_battery_line_state := 'battery_line_on';
		ips_a2_battery_arrow_state := 'battery_arrow_on';
		mpx_a2_state_string := "От АКБ";
		ips1_2_state := 2;	
	ELSE	
		IF ((ips_a2_Invertor = 16) AND (ips_a2_state_reg = 3) AND (ips_a2_inv_byp = 13)) THEN	
			ips_a2_bypass_line_state := 'bypass_line_on';
			ips_a2_bypass_arrow_state := 'bypass_arrow_on';
			ips_a2_input_state := 'arrow_off';
			ips_a2_output_state := 'arrow_on';
			ips_a2_arrow_state := 'arrow_off';
			ips_a2_battery_line_state := 'battery_line_off';
			ips_a2_battery_arrow_state := 'battery_arrow_off';
			mpx_a2_state_string := "Байпас";
			ips1_2_state := 3;	
		ELSE	
			IF ((ips_a2_Invertor = 14) AND (ips_a2_state_reg = 2) AND (ips_a2_inv_byp = 13)) THEN	
				ips_a2_bypass_line_state := 'bypass_line_on';
				ips_a2_bypass_arrow_state := 'bypass_arrow_on';
				ips_a2_input_state := 'arrow_off';
				ips_a2_output_state := 'arrow_on';
				ips_a2_arrow_state := 'arrow_off';
				ips_a2_battery_line_state := 'battery_line_off';
				ips_a2_battery_arrow_state := 'battery_arrow_off';
				mpx_a2_state_string := "Байпас";
				ips1_2_state := 3;	
			ELSE	
				ips_a2_bypass_line_state := 'bypass_line1_off';
				ips_a2_bypass_arrow_state := 'bypass_arrow_off';
				ips_a2_input_state := 'arrow_off';
				ips_a2_output_state := 'arrow_off';
				ips_a2_arrow_state := 'arrow_off';
				ips_a2_battery_line_state := 'battery_line_off';
				ips_a2_battery_arrow_state := 'battery_arrow_off';
				mpx_a2_state_string := "Неизвестно";
				ips1_2_state := 0;
			END_IF
		END_IF
	END_IF
END_IF



IF ((ips_a2_overtemp = 14) OR (ips_a2_overload = 14) OR (ips_a2_outfail = 14) OR (ips_a2_emergency = 14)) THEN
	ips_a2_alarm := TRUE;
ELSE
	ips_a2_alarm := FALSE;
END_IF


//------------------------------------IPS 2.1-------------------------------------
//Конвертация параметров IPS 2.1
ips_s1_in_v_1_real 	 		   	:= ips_s1_in_v_1 * 0.1;
ips_s1_in_v_2_real 	 			:= ips_s1_in_v_2 * 0.1;   		
ips_s1_in_v_3_real 	 		 	:= ips_s1_in_v_3 * 0.1;  		
ips_s1_in_freq_real               := ips_s1_in_freq * 0.1;

ips_s1_bypass_v_1_real			:= ips_s1_bypass_v_1 * 0.1;
ips_s1_bypass_v_2_real			:= ips_s1_bypass_v_2 * 0.1;
ips_s1_bypass_v_3_real			:= ips_s1_bypass_v_3 * 0.1;
ips_s1_bypass_freq_real           := ips_s1_bypass_freq * 0.1;

ips_s1_output_v_1_real			:= ips_s1_output_v_1 * 0.1;
ips_s1_output_v_2_real			:= ips_s1_output_v_2 * 0.1;
ips_s1_output_v_3_real			:= ips_s1_output_v_3 * 0.1;
ips_s1_output_freq_real           := ips_s1_output_freq * 0.1;

ips_s1_load_ph_1_real				:= ips_s1_load_ph_1 * 0.1;
ips_s1_load_ph_2_real				:= ips_s1_load_ph_2 * 0.1;
ips_s1_load_ph_3_real				:= ips_s1_load_ph_3 * 0.1;

ips_s1_output_active_power_1_real	:= ips_s1_power * ips_s1_load_ph_1_real * 0.01 * ips_s1_cosphi;
ips_s1_output_active_power_2_real	:= ips_s1_power * ips_s1_load_ph_2_real * 0.01 * ips_s1_cosphi;
ips_s1_output_active_power_3_real	:= ips_s1_power * ips_s1_load_ph_3_real * 0.01 * ips_s1_cosphi;

ips_s1_output_active_power_1 		:= REAL_TO_WORD(ips_s1_output_active_power_1_real * 1000);
ips_s1_output_active_power_2 		:= REAL_TO_WORD(ips_s1_output_active_power_2_real * 1000);
ips_s1_output_active_power_3 		:= REAL_TO_WORD(ips_s1_output_active_power_3_real * 1000);

ips_s1_battery_voltage_real       := ips_s1_battery_voltage * 1;
ips_s1_battery_current_real       := ips_s1_battery_current * 0.1;

ips_s1_temp_real 					:= ips_s1_temp * 0.1;

//Логика состояний IPS 2.1
IF ((ips_s1_Invertor = 14) AND (ips_s1_state_reg = 2) AND (ips_s1_inv_byp = 12)) THEN
	ips_s1_bypass_line_state := 'bypass_line1_off';
	ips_s1_bypass_arrow_state := 'bypass_arrow_off';
	ips_s1_input_state := 'arrow_on';	
	ips_s1_input_present := TRUE;
	ips_s1_output_state := 'arrow_on';
	ips_s1_arrow_state := 'arrow_on';
	ips_s1_battery_line_state := 'battery_line_on';
	ips_s1_battery_arrow_state := 'battery_arrow_on';
	mpx_s1_state_string := "От сети";	
	ips2_1_state := 1;
ELSE
	IF ((ips_s1_Invertor = 14) AND (ips_s1_state_reg = 3) AND (ips_s1_inv_byp = 12)) THEN	
		ips_s1_bypass_line_state := 'bypass_line1_off';
		ips_s1_bypass_arrow_state := 'bypass_arrow_off';
		ips_s1_input_state := 'arrow_off';
		ips_s1_output_state := 'arrow_on';
		ips_s1_input_present  := FALSE;
		ips_s1_arrow_state := 'arrow_on';
		ips_s1_battery_line_state := 'battery_line_on';
		ips_s1_battery_arrow_state := 'battery_arrow_on';
		mpx_s1_state_string := "От АКБ";
		ips2_1_state := 2;	
	ELSE	
		IF ((ips_s1_Invertor = 16) AND (ips_s1_state_reg = 3) AND (ips_s1_inv_byp = 13)) THEN	
			ips_s1_bypass_line_state := 'bypass_line_on';
			ips_s1_bypass_arrow_state := 'bypass_arrow_on';
			ips_s1_input_state := 'arrow_off';
			ips_s1_input_present := FALSE;
			ips_s1_output_state := 'arrow_on';
			ips_s1_arrow_state := 'arrow_off';
			ips_s1_battery_line_state := 'battery_line_off';
			ips_s1_battery_arrow_state := 'battery_arrow_off';
			mpx_s1_state_string := "Байпас";
			ips2_1_state := 3;	
		ELSE	
			IF ((ips_s1_Invertor = 14) AND (ips_s1_state_reg = 2) AND (ips_s1_inv_byp = 13)) THEN	
				ips_s1_bypass_line_state := 'bypass_line_on';
				ips_s1_bypass_arrow_state := 'bypass_arrow_on';
				ips_s1_input_state := 'arrow_off';
				ips_s1_input_present := FALSE;
				ips_s1_output_state := 'arrow_on';
				ips_s1_arrow_state := 'arrow_off';
				ips_s1_battery_line_state := 'battery_line_off';
				ips_s1_battery_arrow_state := 'battery_arrow_off';
				mpx_s1_state_string := "Байпас";
				ips2_1_state := 3;	
			ELSE	
				ips_s1_bypass_line_state := 'bypass_line1_off';
				ips_s1_bypass_arrow_state := 'bypass_arrow_off';
				ips_s1_input_state := 'arrow_off';
				ips_s1_input_present := FALSE;
				ips_s1_output_state := 'arrow_off';
				ips_s1_arrow_state := 'arrow_off';
				ips_s1_battery_line_state := 'battery_line_off';
				ips_s1_battery_arrow_state := 'battery_arrow_off';
				mpx_s1_state_string := "Неизвестно";
				ips2_1_state := 0;
			END_IF
		END_IF
	END_IF
END_IF


IF ((ips_s1_overtemp = 14) OR (ips_s1_overload = 14) OR (ips_s1_outfail = 14) OR (ips_s1_emergency = 14)) THEN
	ips_s1_alarm := TRUE;
ELSE
	ips_s1_alarm := FALSE;
END_IF

//------------------------------------IPS 2.2-------------------------------------
//Конвертация параметров IPS 2.2
ips_s2_in_v_1_real 	 		   	:= ips_s2_in_v_1 * 0.1;
ips_s2_in_v_2_real 	 			:= ips_s2_in_v_2 * 0.1;   		
ips_s2_in_v_3_real 	 		 	:= ips_s2_in_v_3 * 0.1;  		
ips_s2_in_freq_real               := ips_s2_in_freq * 0.1;

ips_s2_bypass_v_1_real			:= ips_s2_bypass_v_1 * 0.1;
ips_s2_bypass_v_2_real			:= ips_s2_bypass_v_2 * 0.1;
ips_s2_bypass_v_3_real			:= ips_s2_bypass_v_3 * 0.1;
ips_s2_bypass_freq_real           := ips_s2_bypass_freq * 0.1;

ips_s2_output_v_1_real			:= ips_s2_output_v_1 * 0.1;
ips_s2_output_v_2_real			:= ips_s2_output_v_2 * 0.1;
ips_s2_output_v_3_real			:= ips_s2_output_v_3 * 0.1;
ips_s2_output_freq_real           := ips_s2_output_freq * 0.1;

ips_s2_load_ph_1_real				:= ips_s2_load_ph_1 * 0.1;
ips_s2_load_ph_2_real				:= ips_s2_load_ph_2 * 0.1;
ips_s2_load_ph_3_real				:= ips_s2_load_ph_3 * 0.1;

ips_s2_output_active_power_1_real	:= ips_s2_power * ips_s2_load_ph_1_real * 0.01 * ips_s2_cosphi;
ips_s2_output_active_power_2_real	:= ips_s2_power * ips_s2_load_ph_2_real * 0.01 * ips_s2_cosphi;
ips_s2_output_active_power_3_real	:= ips_s2_power * ips_s2_load_ph_3_real * 0.01 * ips_s2_cosphi;

ips_s2_output_active_power_1 		:= REAL_TO_WORD(ips_s2_output_active_power_1_real * 1000);
ips_s2_output_active_power_2 		:= REAL_TO_WORD(ips_s2_output_active_power_2_real * 1000);
ips_s2_output_active_power_3 		:= REAL_TO_WORD(ips_s2_output_active_power_3_real * 1000);

ips_s2_output_active_power_real := ips_s2_output_active_power_1_real + ips_s2_output_active_power_2_real + ips_s2_output_active_power_3_real;

ips_s2_battery_voltage_real       := ips_s2_battery_voltage * 1;
ips_s2_battery_current_real       := ips_s2_battery_current * 0.1;

ips_s2_temp_real 					:= ips_s2_temp * 0.1;

//Логика состояний MPX_s2_1
IF ((ips_s2_Invertor = 14) AND (ips_s2_state_reg = 2) AND (ips_s2_inv_byp = 12)) THEN
	ips_s2_bypass_line_state := 'bypass_line1_off';
	ips_s2_bypass_arrow_state := 'bypass_arrow_off';
	ips_s2_input_state := 'arrow_on';	
	ips_s2_input_present := TRUE;
	ips_s2_output_state := 'arrow_on';
	ips_s2_arrow_state := 'arrow_on';
	ips_s2_battery_line_state := 'battery_line_on';
	ips_s2_battery_arrow_state := 'battery_arrow_on';
	mpx_s2_state_string := "От сети";	
	ips2_2_state := 1;
ELSE
	IF ((ips_s2_Invertor = 14) AND (ips_s2_state_reg = 3) AND (ips_s2_inv_byp = 12)) THEN	
		ips_s2_bypass_line_state := 'bypass_line1_off';
		ips_s2_bypass_arrow_state := 'bypass_arrow_off';
		ips_s2_input_state := 'arrow_off';
		ips_s2_input_present := FALSE;
		ips_s2_output_state := 'arrow_on';
		ips_s2_arrow_state := 'arrow_on';
		ips_s2_battery_line_state := 'battery_line_on';
		ips_s2_battery_arrow_state := 'battery_arrow_on';
		mpx_s2_state_string := "От АКБ";
		ips2_2_state := 2;	
	ELSE	
		IF ((ips_s2_Invertor = 16) AND (ips_s2_state_reg = 3) AND (ips_s2_inv_byp = 13)) THEN	
			ips_s2_bypass_line_state := 'bypass_line_on';
			ips_s2_bypass_arrow_state := 'bypass_arrow_on';
			ips_s2_input_state := 'arrow_off';
			ips_s2_input_present := FALSE;
			ips_s2_output_state := 'arrow_on';
			ips_s2_arrow_state := 'arrow_off';
			ips_s2_battery_line_state := 'battery_line_off';
			ips_s2_battery_arrow_state := 'battery_arrow_off';
			mpx_s2_state_string := "Байпас";
			ips2_2_state := 3;	
		ELSE	
			IF ((ips_s2_Invertor = 14) AND (ips_s2_state_reg = 2) AND (ips_s2_inv_byp = 13)) THEN	
				ips_s2_bypass_line_state := 'bypass_line_on';
				ips_s2_bypass_arrow_state := 'bypass_arrow_on';
				ips_s2_input_state := 'arrow_off';
				ips_s2_input_present := FALSE;
				ips_s2_output_state := 'arrow_on';
				ips_s2_arrow_state := 'arrow_off';
				ips_s2_battery_line_state := 'battery_line_off';
				ips_s2_battery_arrow_state := 'battery_arrow_off';
				mpx_s2_state_string := "Байпас";
				ips2_2_state := 3;	
			ELSE	
				ips_s2_bypass_line_state := 'bypass_line1_off';
				ips_s2_bypass_arrow_state := 'bypass_arrow_off';
				ips_s2_input_state := 'arrow_off';
				ips_s2_input_present := FALSE;
				ips_s2_output_state := 'arrow_off';
				ips_s2_arrow_state := 'arrow_off';
				ips_s2_battery_line_state := 'battery_line_off';
				ips_s2_battery_arrow_state := 'battery_arrow_off';
				mpx_s2_state_string := "Неизвестно";
				ips2_2_state := 0;
			END_IF
		END_IF
	END_IF
END_IF



IF ((ips_s2_overtemp = 14) OR (ips_s2_overload = 14) OR (ips_s2_outfail = 14) OR (ips_s2_emergency = 14)) THEN
	ips_s2_alarm := TRUE;
ELSE
	ips_s2_alarm := FALSE;
END_IF

END_PROGRAM

// CODESYS_Control_for_Raspberry_Pi/Application/GPIO_HANDLER
PROGRAM GPIO_HANDLER
VAR
	
	IN_1: BOOL; // ШОПС: Нарушение ШОС	
	IN_2: BOOL; // ШОПС: Пожар
	IN_3: BOOL; // ШОПС: Неисправность ШОС	
	IN_4: BOOL; // ШАСН: Наличие напряжения на 1 вводе	
	IN_5: BOOL; // ШАСН: Наличие напряжения на 2 вводе	
	IN_6: BOOL; // ШАСН: Наличие напряжения на шине БП
	IN_7: BOOL; // ШАСН: Наличие напряжения на шине ГП
	IN_8: BOOL; // ШАСН: Обогрев в УГП включен	
	IN_9: BOOL; // ШАСН: QS1 в первом положении	
	IN_10: BOOL; // ШАСН: QS1 во втором положении
	IN_11: BOOL; // ШАСН: QFV1 включен
	IN_12: BOOL;  // ШАСН: QFV2 включен
	
	RAW_IN_1: BOOL;
	RAW_IN_2: BOOL;
	RAW_IN_3: BOOL; 
	RAW_IN_4: BOOL; 
	RAW_IN_5: BOOL; 
	RAW_IN_6: BOOL; 
	RAW_IN_7: BOOL; 
	RAW_IN_8: BOOL;
	RAW_IN_9: BOOL;
	RAW_IN_10: BOOL;
	RAW_IN_11: BOOL;
	RAW_IN_12: BOOL; 
END_VAR

 IN_1 := NOT(RAW_IN_1);
 IN_2 := NOT(RAW_IN_2);
 IN_3 := NOT(RAW_IN_3);
 IN_4 := NOT(RAW_IN_4);
 IN_5 := NOT(RAW_IN_5);
 IN_6 := NOT(RAW_IN_6);
 IN_7 := NOT(RAW_IN_7);
 IN_8 := NOT(RAW_IN_8);
 IN_9 := NOT(RAW_IN_9);
 IN_10 := NOT(RAW_IN_10);
 IN_11 := NOT(RAW_IN_11);
 IN_12 := NOT(RAW_IN_12);

END_PROGRAM

// CODESYS_Control_for_Raspberry_Pi/Application/AlarmChecker
PROGRAM AlarmChecker
VAR
	MIN_VOLTAGE : WORD := 50;
	
	ups_s1_in_v_alarm : BOOL;
	ups_s2_in_v_alarm : BOOL;
	ups_a1_in_v_alarm : BOOL;
	ups_a2_in_v_alarm : BOOL;
	
	ups_s1_out_v_alarm : BOOL;
	ups_s2_out_v_alarm : BOOL;
	ups_a1_out_v_alarm : BOOL;
	ups_a2_out_v_alarm : BOOL;
	
	shasn_alarm        : BOOL;
	schrpa_alarm       : BOOL;
	schrps_alarm       : BOOL;
	
	schrps_alarm_raw       	: BOOL;
	Shrps_delay_timer		: TON;

	delay_timeout 			: TIME := T#6S;
	
	shrpa_in_1_alarm	: BOOL;
	shrpa_in_2_alarm	: BOOL;
	shrpa_out_alarm		: BOOL;
	
	shrps_in_1_alarm	: BOOL;
	shrps_in_2_alarm	: BOOL;
	shrps_out_alarm		: BOOL;
	shrps_out_alarm_raw	: BOOL;
END_VAR

//Авария входного напряжения ИБПС1
IF( (PLC_PRG.ips_s1_in_v_1 < MIN_VOLTAGE) OR (PLC_PRG.ips_s1_in_v_2 < MIN_VOLTAGE) OR (PLC_PRG.ips_s1_in_v_3 < MIN_VOLTAGE) OR (PLC_PRG.ips_s1_input_present = FALSE)) THEN
	ups_s1_in_v_alarm := TRUE;
ELSE
	ups_s1_in_v_alarm := FALSE;
END_IF

//Авария входного напряжения ИБПС2
IF((PLC_PRG.ips_s2_in_v_1 < MIN_VOLTAGE) OR (PLC_PRG.ips_s2_in_v_2 < MIN_VOLTAGE) OR (PLC_PRG.ips_s2_in_v_3 < MIN_VOLTAGE) OR (PLC_PRG.ips_s2_input_present = FALSE)) THEN
	ups_s2_in_v_alarm := TRUE;
ELSE
	ups_s2_in_v_alarm := FALSE;
END_IF

//Авария входного напряжения ИБПА1
IF( (PLC_PRG.ips_a1_in_v_1 < MIN_VOLTAGE) OR (PLC_PRG.ips_a1_in_v_2 < MIN_VOLTAGE) OR (PLC_PRG.ips_a1_in_v_3 < MIN_VOLTAGE)) THEN
	ups_a1_in_v_alarm := TRUE;
ELSE
	ups_a1_in_v_alarm := FALSE;
END_IF

//Авария входного напряжения ИБПА2
IF( (PLC_PRG.ips_a2_in_v_1 < MIN_VOLTAGE) OR (PLC_PRG.ips_a2_in_v_2 < MIN_VOLTAGE) OR (PLC_PRG.ips_a2_in_v_3 < MIN_VOLTAGE)) THEN
	ups_a2_in_v_alarm := TRUE;
ELSE
	ups_a2_in_v_alarm := FALSE;
END_IF

//------------------------------------------------------------------------------

//Авария выходного напряжения ИБПС1
IF( (PLC_PRG.ips_s1_output_v_1 < MIN_VOLTAGE) OR (PLC_PRG.ips_s1_output_v_2 < MIN_VOLTAGE) OR (PLC_PRG.ips_s1_output_v_3 < MIN_VOLTAGE)) THEN
	ups_s1_out_v_alarm := TRUE;
ELSE
	ups_s1_out_v_alarm := FALSE;
END_IF

//Авария выходного напряжения ИБПС2
IF( (PLC_PRG.ips_s2_output_v_1 < MIN_VOLTAGE) OR (PLC_PRG.ips_s2_output_v_2 < MIN_VOLTAGE) OR (PLC_PRG.ips_s2_output_v_3 < MIN_VOLTAGE)) THEN
	ups_s2_out_v_alarm := TRUE;
ELSE
	ups_s2_out_v_alarm := FALSE;
END_IF

//Авария выходного напряжения ИБПА1
IF( (PLC_PRG.ips_a1_output_v_1 < MIN_VOLTAGE)) THEN
	ups_a1_out_v_alarm := TRUE;
ELSE
	ups_a1_out_v_alarm := FALSE;
END_IF

//Авария выходного напряжения ИБПА2
IF( (PLC_PRG.ips_a2_output_v_1 < MIN_VOLTAGE)) THEN
	ups_a2_out_v_alarm := TRUE;
ELSE
	ups_a2_out_v_alarm := FALSE;
END_IF

//Авария ШАСН
IF ( (GPIO_HANDLER.IN_4 = FALSE) OR (GPIO_HANDLER.IN_5 = FALSE) ) THEN
	shasn_alarm := TRUE;
ELSE
	shasn_alarm := FALSE;
END_IF

//Авария ЩРПА
IF( (PLC_PRG.shrpa_voltage_1_line_1 < MIN_VOLTAGE) OR (PLC_PRG.shrpa_voltage_1_line_2 < MIN_VOLTAGE) OR (PLC_PRG.shrpa_voltage_1_line_3 < MIN_VOLTAGE) ) THEN
	shrpa_in_1_alarm := TRUE;	
ELSE
	shrpa_in_1_alarm := FALSE;
END_IF

IF( (PLC_PRG.shrpa_voltage_2_line_1 < MIN_VOLTAGE) OR (PLC_PRG.shrpa_voltage_2_line_2 < MIN_VOLTAGE) OR (PLC_PRG.shrpa_voltage_2_line_3 < MIN_VOLTAGE) ) THEN
	shrpa_in_2_alarm := TRUE;	
ELSE
	shrpa_in_2_alarm := FALSE;
END_IF

IF( (PLC_PRG.shrpa_voltage_3_line_1 < MIN_VOLTAGE) OR (PLC_PRG.shrpa_voltage_4_line_1 < MIN_VOLTAGE) ) THEN
	shrpa_out_alarm := TRUE;
ELSE
	shrpa_out_alarm := FALSE;
END_IF

IF ( (shrpa_in_1_alarm = TRUE) OR (shrpa_in_2_alarm = TRUE) OR (shrpa_out_alarm = TRUE) ) THEN
	schrpa_alarm := TRUE;
ELSE
	schrpa_alarm := FALSE;
END_IF

//Авария ЩРПС
IF( PLC_PRG.shrps_voltage_1_line_1 < MIN_VOLTAGE ) THEN
	shrps_in_1_alarm := TRUE;	
ELSE
	shrps_in_1_alarm := FALSE;
END_IF

IF( PLC_PRG.shrps_voltage_2_line_1 < MIN_VOLTAGE ) THEN
	shrps_in_2_alarm := TRUE;	
ELSE
	shrps_in_2_alarm := FALSE;
END_IF

IF ( (PLC_PRG.shrps_ups_bus_1 = FALSE) OR (PLC_PRG.shrps_ups_bus_2 = FALSE) ) THEN
	shrps_out_alarm_raw := TRUE;
ELSE
	shrps_out_alarm_raw := FALSE;
END_IF
Shrps_delay_timer(IN := shrps_out_alarm_raw, PT:= delay_timeout);
shrps_out_alarm :=Shrps_delay_timer.Q;

IF ( (shrps_in_1_alarm = TRUE) OR (shrps_in_2_alarm = TRUE) OR (shrps_out_alarm = TRUE) ) THEN
	schrps_alarm := TRUE;
ELSE
	schrps_alarm := FALSE;
END_IF

END_PROGRAM

// CODESYS_Control_for_Raspberry_Pi/Application/BusReinit
PROGRAM BusReinit
VAR
	BL1 : BLINK;
	BL2 : BLINK;
	BL3 : BLINK;
	BL4 : BLINK;
	BL5 : BLINK;
	BL6 : BLINK;
	BL7 : BLINK;
	BL8 : BLINK;
	BL9 : BLINK;
	BL10 : BLINK;
	BL11 : BLINK;
	BL12 : BLINK;
END_VAR

IF PLC.xError THEN 
	BL1(enable:=TRUE, timelow:=T#50MS, timehigh:=T#100MS);
	PLC.xReset:=BL1.OUT; 
	ModbusMaster.xResetComPort := TRUE;
ELSE 
	BL1(enable:=FALSE, timelow:=T#50MS, timehigh:=T#100MS);
	PLC.xReset:= FALSE;
	ModbusMaster.xResetComPort := FALSE; 
END_IF;

IF SHRPA_ICP_CON.xError THEN 
	BL2(enable:=TRUE, timelow:=T#50MS, timehigh:=T#100MS);
	SHRPA_ICP_CON.xReset:=BL2.OUT; 
	ModbusMaster.xResetComPort := TRUE;
ELSE 
	BL2(enable:=FALSE, timelow:=T#50MS, timehigh:=T#100MS);
	SHRPA_ICP_CON.xReset:= FALSE;
	ModbusMaster.xResetComPort := FALSE; 
END_IF;

IF SHRPS_ICP_CON.xError THEN 
	BL3(enable:=TRUE, timelow:=T#50MS, timehigh:=T#100MS);
	SHRPS_ICP_CON.xReset:=BL3.OUT; 
	ModbusMaster.xResetComPort := TRUE;
ELSE 
	BL3(enable:=FALSE, timelow:=T#50MS, timehigh:=T#100MS);
	SHRPS_ICP_CON.xReset:= FALSE;
	ModbusMaster.xResetComPort := FALSE; 
END_IF;

IF SHASN_ICP_CON.xError THEN 
	BL4(enable:=TRUE, timelow:=T#50MS, timehigh:=T#100MS);
	SHASN_ICP_CON.xReset:=BL4.OUT; 
	ModbusMaster.xResetComPort := TRUE;
ELSE 
	BL4(enable:=FALSE, timelow:=T#50MS, timehigh:=T#100MS);
	SHASN_ICP_CON.xReset:= FALSE;
	ModbusMaster.xResetComPort := FALSE; 
END_IF;

IF SHRPA_ELNET_1.xError THEN 
	BL5(enable:=TRUE, timelow:=T#50MS, timehigh:=T#100MS);
	SHRPA_ELNET_1.xReset:=BL5.OUT; 
	ModbusMaster.xResetComPort := TRUE;
ELSE 
	BL5(enable:=FALSE, timelow:=T#50MS, timehigh:=T#100MS);
	SHRPA_ELNET_1.xReset:= FALSE;
	ModbusMaster.xResetComPort := FALSE; 
END_IF;

IF SHRPA_ELNET_2.xError THEN 
	BL6(enable:=TRUE, timelow:=T#50MS, timehigh:=T#100MS);
	SHRPA_ELNET_2.xReset:=BL6.OUT; 
	ModbusMaster.xResetComPort := TRUE;
ELSE 
	BL6(enable:=FALSE, timelow:=T#50MS, timehigh:=T#100MS);
	SHRPA_ELNET_2.xReset:= FALSE;
	ModbusMaster.xResetComPort := FALSE; 
END_IF;

IF SHRPA_ELNET_3.xError THEN 
	BL7(enable:=TRUE, timelow:=T#50MS, timehigh:=T#100MS);
	SHRPA_ELNET_3.xReset:=BL7.OUT; 
	ModbusMaster.xResetComPort := TRUE;
ELSE 
	BL7(enable:=FALSE, timelow:=T#50MS, timehigh:=T#100MS);
	SHRPA_ELNET_3.xReset:= FALSE;
	ModbusMaster.xResetComPort := FALSE; 
END_IF;

IF SHRPA_ELNET_4.xError THEN 
	BL8(enable:=TRUE, timelow:=T#50MS, timehigh:=T#100MS);
	SHRPA_ELNET_4.xReset:=BL8.OUT; 
	ModbusMaster.xResetComPort := TRUE;
ELSE 
	BL8(enable:=FALSE, timelow:=T#50MS, timehigh:=T#100MS);
	SHRPA_ELNET_4.xReset:= FALSE;
	ModbusMaster.xResetComPort := FALSE; 
END_IF;

IF SHRPS_ELNET_1.xError THEN 
	BL9(enable:=TRUE, timelow:=T#50MS, timehigh:=T#100MS);
	SHRPS_ELNET_1.xReset:=BL9.OUT; 
	ModbusMaster.xResetComPort := TRUE;
ELSE 
	BL9(enable:=FALSE, timelow:=T#50MS, timehigh:=T#100MS);
	SHRPS_ELNET_1.xReset:= FALSE;
	ModbusMaster.xResetComPort := FALSE; 
END_IF;

IF SHRPS_ELNET_2.xError THEN 
	BL10(enable:=TRUE, timelow:=T#50MS, timehigh:=T#100MS);
	SHRPS_ELNET_2.xReset:=BL10.OUT; 
	ModbusMaster.xResetComPort := TRUE;
ELSE 
	BL10(enable:=FALSE, timelow:=T#50MS, timehigh:=T#100MS);
	SHRPS_ELNET_2.xReset:= FALSE;
	ModbusMaster.xResetComPort := FALSE; 
END_IF;

IF SHRPS_ELNET_3.xError THEN 
	BL11(enable:=TRUE, timelow:=T#50MS, timehigh:=T#100MS);
	SHRPS_ELNET_3.xReset:=BL11.OUT; 
	ModbusMaster.xResetComPort := TRUE;
ELSE 
	BL11(enable:=FALSE, timelow:=T#50MS, timehigh:=T#100MS);
	SHRPS_ELNET_3.xReset:= FALSE;
	ModbusMaster.xResetComPort := FALSE; 
END_IF;

IF SHRPS_ELNET_4.xError THEN 
	BL12(enable:=TRUE, timelow:=T#50MS, timehigh:=T#100MS);
	SHRPS_ELNET_4.xReset:=BL12.OUT; 
	ModbusMaster.xResetComPort := TRUE;
ELSE 
	BL12(enable:=FALSE, timelow:=T#50MS, timehigh:=T#100MS);
	SHRPS_ELNET_4.xReset:= FALSE;
	ModbusMaster.xResetComPort := FALSE; 
END_IF;

END_PROGRAM

// CODESYS_Control_for_Raspberry_Pi/Application/visualization/monitoring
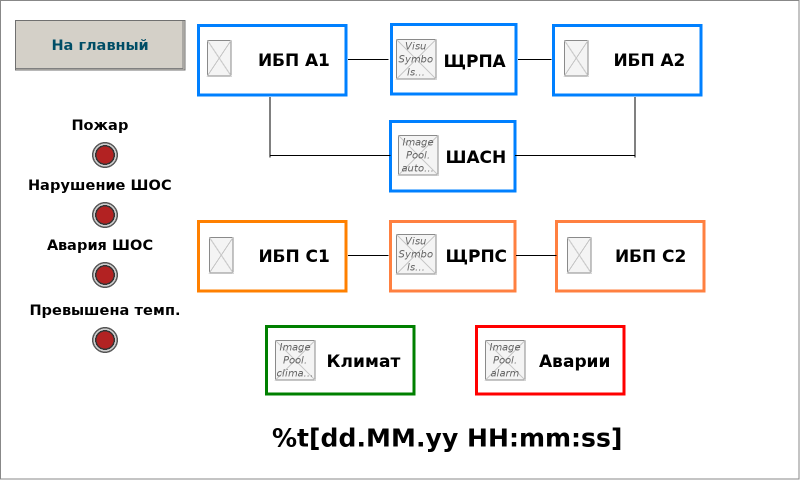
VISUALIZATION monitoring  // 800x480, background image ImagePool.bg_800
    Lamp1 (90,140 30x30), variable: GPIO_HANDLER.IN_2, style: Lamp-Lamp1-Red
    Rectangle (20,110 160x30), "Пожар"
    Lamp1 (90,200 30x30), variable: GPIO_HANDLER.IN_1, style: Lamp-Lamp1-Red
    Rectangle (20,170 160x30), "Нарушение ШОС"
    Lamp1 (90,260 30x30), variable: GPIO_HANDLER.IN_3, style: Lamp-Lamp1-Red
    Rectangle (20,230 160x30), "Авария ШОС"
    Lamp1 (90,325 30x30), variable: PLC_PRG.climate_temp_excess, style: Lamp-Lamp1-Red
    Rectangle (20,295 170x30), "Превышена темп."
    RoundedRectangle (389,220 127x72), colour toggle: AlarmChecker.schrps_alarm
        OnMouseClick:  Assign=schrps, Type=Assignment
    Group (396,234 118x40)
        RoundedRectangle (43,6 75x32), "ЩРПС"
            OnMouseClick:  Assign=schrps, Type=Assignment
        Image (0,0 40x40), image: VisuSymbols.Symbols.TreeDown
    Group (390,23 127x72)
        OnMouseClick:  Assign=schrpa, Type=Assignment
        RoundedRectangle (0,0 127x72), colour toggle: AlarmChecker.schrpa_alarm
            OnMouseClick:  Assign=schrpa, Type=Assignment
        Image (6,16 40x40), image: VisuSymbols.Symbols.TreeDown
        RoundedRectangle (52,22 65x32), "ЩРПА"
            OnMouseClick:  Assign=schrpa, Type=Assignment
    Group (389,120 127x72)
        OnMouseClick:  Assign=shasn, Type=Assignment
        RoundedRectangle (0,0 127x72), colour toggle: AlarmChecker.shasn_alarm
            OnMouseClick:  Assign=shasn, Type=Assignment
        RoundedRectangle (48,21 78x32), "ШАСН"
            OnMouseClick:  Assign=shasn, Type=Assignment
        Image (9,15 40x40), image: ImagePool.automation-512
    Button (15,20 170x50), "На главный"
        OnMouseClick:  Assign=main, Type=Assignment
    Group (265,325 150x70)
        OnMouseClick:  Assign=climate, Type=Assignment
        RoundedRectangle (0,0 150x70)
            OnMouseClick:  Assign=climate, Type=Assignment
        RoundedRectangle (55,20 87x32), "Климат"
            OnMouseClick:  Assign=climate, Type=Assignment
        Image (10,15 40x40), image: ImagePool.climate
    Group (475,325 150x70)
        OnMouseClick:  Assign=alarm, Type=Assignment
        RoundedRectangle (0,0 150x70)
            OnMouseClick:  Assign=alarm, Type=Assignment
        RoundedRectangle (55,20 90x32), "Аварии"
            OnMouseClick:  Assign=alarm, Type=Assignment
        Image (10,15 40x40), image: ImagePool.alarm
    Group (197,220 150x72)
        OnMouseClick:  Assign=ups_s1_state, Type=Assignment
        RoundedRectangle (0,0 150x72), colour toggle: AlarmChecker.ups_s1_in_v_alarm
        RoundedRectangle (48,20 99x32), "ИБП С1"
            OnMouseClick:  Assign=ups_s1_params, Type=Assignment
        Image (12,17 24x36), image: ImagePool.mini_ups
    Group (555,220 150x72)
        OnMouseClick:  Assign=ups_s2_state, Type=Assignment
        RoundedRectangle (0,0 150x72), colour toggle: AlarmChecker.ups_s2_in_v_alarm
        RoundedRectangle (45,20 102x32), "ИБП С2"
            OnMouseClick:  Assign=ups_s2_params, Type=Assignment
        Image (12,17 24x36), image: ImagePool.mini_ups
    Group (197,24 150x72)
        OnMouseClick:  Assign=ups_a1_state, Type=Assignment
        RoundedRectangle (0,0 150x72), colour toggle: AlarmChecker.ups_a1_in_v_alarm
            OnMouseClick:  Assign=ups_a1_state, Type=Assignment
        RoundedRectangle (50,20 94x32), "ИБП А1"
        Image (10,16 24x36), image: ImagePool.mini_ups
    Rectangle (260,415 375x45), "%t[dd.MM.yy HH:mm:ss]"
    Group (552,24 150x72)
        OnMouseClick:  Assign=ups_a2_state, Type=Assignment
        RoundedRectangle (0,0 150x72), colour toggle: AlarmChecker.ups_a2_in_v_alarm
            OnMouseClick:  Assign=ups_a2_state, Type=Assignment
        RoundedRectangle (48,20 99x32), "ИБП А2"
        Image (12,16 24x36), image: ImagePool.mini_ups
    Line (640,130)
    Line (635,157) (635,97)
    Line (515,155) (635,155)
    Line (270,155) (390,155)
    Line (270,157) (270,97)
    Line (348,59) (388,59)
    Line (518,59) (551,59)
    Line (348,255) (388,255)
    Line (516,255) (556,255)
    hotkey  Id=481037385728, Key=KeyDown=True, KeyName=0, VisuElemId=148
    hotkey  Id=481038434304, Key=KeyName=0, VisuElemId=148
END_VISUALIZATION

